LIN {X 0,Y 464.947,Z 367.068,A -85,B 0,C 180,E1 22700.512,E2 22700.512} C_VEL
LIN {X 0,Y 464.933,Z 367.036,A -85,B 0,C 180,E1 22696.87,E2 22696.87} C_VEL
LIN {X 0,Y 464.97,Z 367.067,A -85,B 0,C 180,E1 22693.422,E2 22693.422} C_VEL
LIN {X 0,Y 464.989,Z 367.031,A -85,B 0,C 180,E1 22689.774,E2 22689.774} C_VEL
LIN {X 0,Y 464.946,Z 367.064,A -85,B 0,C 180,E1 22686.291,E2 22686.291} C_VEL
LIN {X 0,Y 464.937,Z 367.047,A -85,B 0,C 180,E1 22682.706,E2 22682.706} C_VEL
LIN {X 0,Y 464.965,Z 367.06,A -85,B 0,C 180,E1 22679.132,E2 22679.132} C_VEL
LIN {X 0,Y 464.99,Z 367.048,A -85,B 0,C 180,E1 22675.555,E2 22675.555} C_VEL
LIN {X 0,Y 464.944,Z 367.049,A -85,B 0,C 180,E1 22672.084,E2 22672.084} C_VEL
LIN {X 0,Y 464.94,Z 367.063,A -85,B 0,C 180,E1 22668.459,E2 22668.459} C_VEL
LIN {X 0,Y 464.965,Z 367.041,A -85,B 0,C 180,E1 22664.906,E2 22664.906} C_VEL
LIN {X 0,Y 464.994,Z 367.06,A -85,B 0,C 180,E1 22661.309,E2 22661.309} C_VEL
LIN {X 0,Y 464.95,Z 367.044,A -85,B 0,C 180,E1 22657.756,E2 22657.756} C_VEL
LIN {X 0,Y 464.943,Z 367.064,A -85,B 0,C 180,E1 22654.249,E2 22654.249} C_VEL
LIN {X 0,Y 464.978,Z 367.05,A -85,B 0,C 180,E1 22650.779,E2 22650.779} C_VEL
LIN {X 0,Y 464.984,Z 367.05,A -85,B 0,C 180,E1 22647.219,E2 22647.219} C_VEL
LIN {X 0,Y 464.945,Z 367.068,A -85,B 0,C 180,E1 22643.741,E2 22643.741} C_VEL
LIN {X 0,Y 464.947,Z 367.069,A -85,B 0,C 180,E1 22640.142,E2 22640.142} C_VEL
LIN {X 0,Y 464.987,Z 367.066,A -85,B 0,C 180,E1 22636.617,E2 22636.617} C_VEL
LIN {X 0,Y 464.986,Z 367.052,A -85,B 0,C 180,E1 22632.971,E2 22632.971} C_VEL
LIN {X 0,Y 464.98,Z 367.258,A -85,B 0,C 180,E1 22631.366,E2 22631.366} C_VEL
LIN {X 0,Y 469.561,Z 382.374,A -85,B 0,C 180,E1 22628.405,E2 22628.405} C_VEL
LIN {X 0,Y 472.417,Z 392.249,A -85,B 0,C 180,E1 22626.661,E2 22626.661} C_VEL
LIN {X 0,Y 477.627,Z 402.671,A -85,B 0,C 180,E1 22626.002,E2 22626.002} C_VEL
LIN {X 0,Y 483.965,Z 427.071,A -85,B 0,C 180,E1 22625.03,E2 22625.03} C_VEL
LIN {X 0,Y 480.044,Z 648.164,A -85,B 0,C 180,E1 22621.453,E2 22621.453} C_VEL
LIN {X 0,Y 479.301,Z 666.693,A -85,B 0,C 180,E1 22621.018,E2 22621.018} C_VEL
LIN {X 0,Y 478.11,Z 687.493,A -85,B 0,C 180,E1 22620.307,E2 22620.307} C_VEL
LIN {X 0,Y 476.875,Z 704.905,A -85,B 0,C 180,E1 22619.519,E2 22619.519} C_VEL
LIN {X 0,Y 475.534,Z 721.763,A -85,B 0,C 180,E1 22618.581,E2 22618.581} C_VEL
LIN {X 0,Y 473.78,Z 741.15,A -85,B 0,C 180,E1 22617.254,E2 22617.254} C_VEL
LIN {X 0,Y 472.31,Z 756.498,A -85,B 0,C 180,E1 22615.989,E2 22615.989} C_VEL
LIN {X 0,Y 470.857,Z 771.086,A -85,B 0,C 180,E1 22614.594,E2 22614.594} C_VEL
LIN {X 0,Y 469.132,Z 788.25,A -85,B 0,C 180,E1 22612.65,E2 22612.65} C_VEL
LIN {X 0,Y 467.883,Z 800.978,A -85,B 0,C 180,E1 22610.951,E2 22610.951} C_VEL
LIN {X 0,Y 466.724,Z 813.64,A -85,B 0,C 180,E1 22609.003,E2 22609.003} C_VEL
LIN {X 0,Y 465.696,Z 825.892,A -85,B 0,C 180,E1 22606.745,E2 22606.745} C_VEL
LIN {X 0,Y 465.054,Z 834.762,A -85,B 0,C 180,E1 22604.823,E2 22604.823} C_VEL
LIN {X 0,Y 464.527,Z 843.637,A -85,B 0,C 180,E1 22602.556,E2 22602.556} C_VEL
LIN {X 0,Y 464.18,Z 851.15,A -85,B 0,C 180,E1 22600.129,E2 22600.129} C_VEL
LIN {X 0,Y 464.022,Z 856.246,A -85,B 0,C 180,E1 22598.051,E2 22598.051} C_VEL
LIN {X 0,Y 463.947,Z 860.214,A -85,B 0,C 180,E1 22595.937,E2 22595.937} C_VEL
LIN {X 0,Y 463.913,Z 863.438,A -85,B 0,C 180,E1 22593.336,E2 22593.336} C_VEL
LIN {X 0,Y 463.91,Z 864.696,A -85,B 0,C 180,E1 22591.111,E2 22591.111} C_VEL
LIN {X 0,Y 463.91,Z 864.755,A -85,B 0,C 180,E1 22589.136,E2 22589.136} C_VEL
LIN {X 0,Y 463.914,Z 863.704,A -85,B 0,C 180,E1 22587.035,E2 22587.035} C_VEL
LIN {X 0,Y 463.935,Z 861.041,A -85,B 0,C 180,E1 22584.559,E2 22584.559} C_VEL
LIN {X 0,Y 464.016,Z 856.788,A -85,B 0,C 180,E1 22582.198,E2 22582.198} C_VEL
LIN {X 0,Y 464.154,Z 852.036,A -85,B 0,C 180,E1 22580.202,E2 22580.202} C_VEL
LIN {X 0,Y 464.42,Z 845.709,A -85,B 0,C 180,E1 22578.072,E2 22578.072} C_VEL
LIN {X 0,Y 464.954,Z 836.391,A -85,B 0,C 180,E1 22575.555,E2 22575.555} C_VEL
LIN {X 0,Y 465.589,Z 827.257,A -85,B 0,C 180,E1 22573.533,E2 22573.533} C_VEL
LIN {X 0,Y 466.4,Z 817.262,A -85,B 0,C 180,E1 22571.632,E2 22571.632} C_VEL
LIN {X 0,Y 467.614,Z 803.952,A -85,B 0,C 180,E1 22569.473,E2 22569.473} C_VEL
LIN {X 0,Y 468.852,Z 790.947,A -85,B 0,C 180,E1 22567.692,E2 22567.692} C_VEL
LIN {X 0,Y 470.182,Z 777.792,A -85,B 0,C 180,E1 22566.126,E2 22566.126} C_VEL
LIN {X 0,Y 471.902,Z 760.777,A -85,B 0,C 180,E1 22564.392,E2 22564.392} C_VEL
LIN {X 0,Y 473.431,Z 744.821,A -85,B 0,C 180,E1 22563.033,E2 22563.033} C_VEL
LIN {X 0,Y 474.846,Z 729.536,A -85,B 0,C 180,E1 22561.92,E2 22561.92} C_VEL
LIN {X 0,Y 476.477,Z 710.731,A -85,B 0,C 180,E1 22560.777,E2 22560.777} C_VEL
LIN {X 0,Y 477.784,Z 692.136,A -85,B 0,C 180,E1 22559.887,E2 22559.887} C_VEL
LIN {X 0,Y 478.841,Z 675.18,A -85,B 0,C 180,E1 22559.246,E2 22559.246} C_VEL
LIN {X 0,Y 479.873,Z 654.59,A -85,B 0,C 180,E1 22558.671,E2 22558.671} C_VEL
LIN {X 0,Y 480.66,Z 617.37,A -85,B 0,C 180,E1 22558.034,E2 22558.034} C_VEL
LIN {X 0,Y 483.896,Z 426.069,A -85,B 0,C 180,E1 22554.947,E2 22554.947} C_VEL
LIN {X 0,Y 476.986,Z 401.05,A -85,B 0,C 180,E1 22553.913,E2 22553.913} C_VEL
LIN {X 0,Y 472.254,Z 391.785,A -85,B 0,C 180,E1 22553.289,E2 22553.289} C_VEL
LIN {X 0,Y 467.71,Z 376.233,A -85,B 0,C 180,E1 22550.429,E2 22550.429} C_VEL
LIN {X 0,Y 464.964,Z 367.167,A -85,B 0,C 180,E1 22548.586,E2 22548.586} C_VEL
LIN {X 0,Y 464.988,Z 367.054,A -85,B 0,C 180,E1 22545.031,E2 22545.031} C_VEL
LIN {X 0,Y 464.973,Z 367.053,A -85,B 0,C 180,E1 22541.48,E2 22541.48} C_VEL
LIN {X 0,Y 464.942,Z 367.054,A -85,B 0,C 180,E1 22537.959,E2 22537.959} C_VEL
LIN {X 0,Y 464.946,Z 367.058,A -85,B 0,C 180,E1 22534.297,E2 22534.297} C_VEL
LIN {X 0,Y 464.99,Z 367.066,A -85,B 0,C 180,E1 22530.785,E2 22530.785} C_VEL
LIN {X 0,Y 464.969,Z 367.038,A -85,B 0,C 180,E1 22527.264,E2 22527.264} C_VEL
LIN {X 0,Y 464.941,Z 367.065,A -85,B 0,C 180,E1 22523.716,E2 22523.716} C_VEL
LIN {X 0,Y 464.943,Z 367.055,A -85,B 0,C 180,E1 22519.992,E2 22519.992} C_VEL
LIN {X 0,Y 464.977,Z 367.056,A -85,B 0,C 180,E1 22516.459,E2 22516.459} C_VEL
LIN {X 0,Y 464.964,Z 367.04,A -85,B 0,C 180,E1 22513.054,E2 22513.054} C_VEL
LIN {X 0,Y 464.939,Z 367.066,A -85,B 0,C 180,E1 22509.536,E2 22509.536} C_VEL
LIN {X 0,Y 464.945,Z 367.037,A -85,B 0,C 180,E1 22505.93,E2 22505.93} C_VEL
LIN {X 0,Y 464.988,Z 367.066,A -85,B 0,C 180,E1 22502.347,E2 22502.347} C_VEL
LIN {X 0,Y 464.954,Z 367.035,A -85,B 0,C 180,E1 22498.896,E2 22498.896} C_VEL
LIN {X 0,Y 464.94,Z 367.065,A -85,B 0,C 180,E1 22495.318,E2 22495.318} C_VEL
LIN {X 0,Y 464.948,Z 367.043,A -85,B 0,C 180,E1 22491.722,E2 22491.722} C_VEL
LIN {X 0,Y 464.992,Z 367.054,A -85,B 0,C 180,E1 22488.219,E2 22488.219} C_VEL
LIN {X 0,Y 464.957,Z 367.054,A -85,B 0,C 180,E1 22484.669,E2 22484.669} C_VEL
LIN {X 0,Y 464.936,Z 367.06,A -85,B 0,C 180,E1 22481.121,E2 22481.121} C_VEL
LIN {X 0,Y 464.948,Z 367.053,A -85,B 0,C 180,E1 22477.501,E2 22477.501} C_VEL
LIN {X 0,Y 464.992,Z 367.055,A -85,B 0,C 180,E1 22473.99,E2 22473.99} C_VEL
LIN {X 0,Y 464.954,Z 367.067,A -85,B 0,C 180,E1 22470.507,E2 22470.507} C_VEL
LIN {X 0,Y 464.937,Z 367.068,A -85,B 0,C 180,E1 22466.9,E2 22466.9} C_VEL
LIN {X 0,Y 464.95,Z 367.067,A -85,B 0,C 180,E1 22463.295,E2 22463.295} C_VEL
LIN {X 0,Y 464.999,Z 367.064,A -85,B 0,C 180,E1 22459.757,E2 22459.757} C_VEL
LIN {X 0,Y 464.968,Z 367.069,A -85,B 0,C 180,E1 22456.084,E2 22456.084} C_VEL
LIN {X 0,Y 464.936,Z 367.069,A -85,B 0,C 180,E1 22452.64,E2 22452.64} C_VEL
LIN {X 0,Y 464.948,Z 367.067,A -85,B 0,C 180,E1 22449.055,E2 22449.055} C_VEL
LIN {X 0,Y 464.987,Z 367.065,A -85,B 0,C 180,E1 22445.49,E2 22445.49} C_VEL
LIN {X 0,Y 464.965,Z 367.067,A -85,B 0,C 180,E1 22441.87,E2 22441.87} C_VEL
LIN {X 0,Y 464.937,Z 367.068,A -85,B 0,C 180,E1 22438.376,E2 22438.376} C_VEL
LIN {X 0,Y 464.939,Z 367.07,A -85,B 0,C 180,E1 22434.657,E2 22434.657} C_VEL
LIN {X 0,Y 464.983,Z 367.067,A -85,B 0,C 180,E1 22431.176,E2 22431.176} C_VEL
LIN {X 0,Y 464.972,Z 367.067,A -85,B 0,C 180,E1 22429.595,E2 22429.595} C_VEL
LIN {X 0,Y 464.033,Z 367.192,A -85,B 0,C 180,E1 22428.646,E2 22428.646} C_VEL
LIN {X 0,Y 457.477,Z 368.001,A -85,B 0,C 180,E1 22425.906,E2 22425.906} C_VEL
LIN {X 0,Y 457.055,Z 368.052,A -85,B 0,C 180,E1 22425.278,E2 22425.278} C_VEL
LIN {X 0,Y 457.018,Z 368.057,A -85,B 0,C 180,E1 22421.611,E2 22421.611} C_VEL
LIN {X 0,Y 456.994,Z 368.06,A -85,B 0,C 180,E1 22418.049,E2 22418.049} C_VEL
LIN {X 0,Y 457.001,Z 368.057,A -85,B 0,C 180,E1 22414.392,E2 22414.392} C_VEL
LIN {X 0,Y 457.045,Z 368.053,A -85,B 0,C 180,E1 22410.877,E2 22410.877} C_VEL
LIN {X 0,Y 457.028,Z 368.055,A -85,B 0,C 180,E1 22407.241,E2 22407.241} C_VEL
LIN {X 0,Y 456.996,Z 368.059,A -85,B 0,C 180,E1 22403.72,E2 22403.72} C_VEL
LIN {X 0,Y 456.997,Z 368.059,A -85,B 0,C 180,E1 22400.047,E2 22400.047} C_VEL
LIN {X 0,Y 457.027,Z 368.055,A -85,B 0,C 180,E1 22396.463,E2 22396.463} C_VEL
LIN {X 0,Y 457.04,Z 368.054,A -85,B 0,C 180,E1 22392.911,E2 22392.911} C_VEL
LIN {X 0,Y 457.001,Z 368.056,A -85,B 0,C 180,E1 22389.376,E2 22389.376} C_VEL
LIN {X 0,Y 456.997,Z 368.059,A -85,B 0,C 180,E1 22385.713,E2 22385.713} C_VEL
LIN {X 0,Y 457.017,Z 368.057,A -85,B 0,C 180,E1 22382.084,E2 22382.084} C_VEL
LIN {X 0,Y 457.055,Z 368.054,A -85,B 0,C 180,E1 22378.541,E2 22378.541} C_VEL
LIN {X 0,Y 457.019,Z 368.057,A -85,B 0,C 180,E1 22374.874,E2 22374.874} C_VEL
LIN {X 0,Y 456.997,Z 368.057,A -85,B 0,C 180,E1 22371.265,E2 22371.265} C_VEL
LIN {X 0,Y 457.006,Z 368.058,A -85,B 0,C 180,E1 22367.636,E2 22367.636} C_VEL
LIN {X 0,Y 457.042,Z 368.055,A -85,B 0,C 180,E1 22364.07,E2 22364.07} C_VEL
LIN {X 0,Y 457.048,Z 368.054,A -85,B 0,C 180,E1 22360.346,E2 22360.346} C_VEL
LIN {X 0,Y 457.005,Z 368.056,A -85,B 0,C 180,E1 22356.8,E2 22356.8} C_VEL
LIN {X 0,Y 456.999,Z 368.058,A -85,B 0,C 180,E1 22353.15,E2 22353.15} C_VEL
LIN {X 0,Y 457.025,Z 368.056,A -85,B 0,C 180,E1 22349.624,E2 22349.624} C_VEL
LIN {X 0,Y 457.049,Z 368.045,A -85,B 0,C 180,E1 22346.078,E2 22346.078} C_VEL
LIN {X 0,Y 457.01,Z 368.042,A -85,B 0,C 180,E1 22342.504,E2 22342.504} C_VEL
LIN {X 0,Y 456.998,Z 368.048,A -85,B 0,C 180,E1 22338.886,E2 22338.886} C_VEL
LIN {X 0,Y 457.011,Z 368.044,A -85,B 0,C 180,E1 22335.247,E2 22335.247} C_VEL
LIN {X 0,Y 457.053,Z 368.041,A -85,B 0,C 180,E1 22331.732,E2 22331.732} C_VEL
LIN {X 0,Y 457.025,Z 368.031,A -85,B 0,C 180,E1 22328.043,E2 22328.043} C_VEL
LIN {X 0,Y 457.001,Z 368.054,A -85,B 0,C 180,E1 22324.512,E2 22324.512} C_VEL
LIN {X 0,Y 456.999,Z 368.028,A -85,B 0,C 180,E1 22320.747,E2 22320.747} C_VEL
LIN {X 0,Y 457.039,Z 368.053,A -85,B 0,C 180,E1 22317.236,E2 22317.236} C_VEL
LIN {X 0,Y 457.046,Z 368.017,A -85,B 0,C 180,E1 22313.589,E2 22313.589} C_VEL
LIN {X 0,Y 457.009,Z 368.055,A -85,B 0,C 180,E1 22310.042,E2 22310.042} C_VEL
LIN {X 0,Y 457,Z 368.027,A -85,B 0,C 180,E1 22306.457,E2 22306.457} C_VEL
LIN {X 0,Y 457.034,Z 368.056,A -85,B 0,C 180,E1 22302.941,E2 22302.941} C_VEL
LIN {X 0,Y 457.058,Z 368.022,A -85,B 0,C 180,E1 22299.24,E2 22299.24} C_VEL
LIN {X 0,Y 457.015,Z 368.055,A -85,B 0,C 180,E1 22295.709,E2 22295.709} C_VEL
LIN {X 0,Y 457,Z 368.026,A -85,B 0,C 180,E1 22292.078,E2 22292.078} C_VEL
LIN {X 0,Y 457.017,Z 368.053,A -85,B 0,C 180,E1 22288.47,E2 22288.47} C_VEL
LIN {X 0,Y 457.052,Z 368.052,A -85,B 0,C 180,E1 22284.872,E2 22284.872} C_VEL
LIN {X 0,Y 457.032,Z 368.045,A -85,B 0,C 180,E1 22281.264,E2 22281.264} C_VEL
LIN {X 0,Y 457.006,Z 368.05,A -85,B 0,C 180,E1 22277.686,E2 22277.686} C_VEL
LIN {X 0,Y 457.006,Z 368.061,A -85,B 0,C 180,E1 22273.91,E2 22273.91} C_VEL
LIN {X 0,Y 457.037,Z 368.25,A -85,B 0,C 180,E1 22272.022,E2 22272.022} C_VEL
LIN {X 0,Y 461.532,Z 382.762,A -85,B 0,C 180,E1 22269.08,E2 22269.08} C_VEL
LIN {X 0,Y 464.235,Z 391.951,A -85,B 0,C 180,E1 22267.416,E2 22267.416} C_VEL
LIN {X 0,Y 471.676,Z 406.668,A -85,B 0,C 180,E1 22266.451,E2 22266.451} C_VEL
LIN {X 0,Y 477.373,Z 428.874,A -85,B 0,C 180,E1 22265.549,E2 22265.549} C_VEL
LIN {X 0,Y 473.204,Z 648.338,A -85,B 0,C 180,E1 22261.952,E2 22261.952} C_VEL
LIN {X 0,Y 472.379,Z 667.608,A -85,B 0,C 180,E1 22261.49,E2 22261.49} C_VEL
LIN {X 0,Y 471.092,Z 688.176,A -85,B 0,C 180,E1 22260.763,E2 22260.763} C_VEL
LIN {X 0,Y 469.847,Z 704.666,A -85,B 0,C 180,E1 22260.005,E2 22260.005} C_VEL
LIN {X 0,Y 468.407,Z 721.599,A -85,B 0,C 180,E1 22259.052,E2 22259.052} C_VEL
LIN {X 0,Y 466.547,Z 740.909,A -85,B 0,C 180,E1 22257.713,E2 22257.713} C_VEL
LIN {X 0,Y 464.968,Z 756.256,A -85,B 0,C 180,E1 22256.431,E2 22256.431} C_VEL
LIN {X 0,Y 463.362,Z 771.413,A -85,B 0,C 180,E1 22254.958,E2 22254.958} C_VEL
LIN {X 0,Y 461.598,Z 787.697,A -85,B 0,C 180,E1 22253.082,E2 22253.082} C_VEL
LIN {X 0,Y 460.272,Z 800.136,A -85,B 0,C 180,E1 22251.404,E2 22251.404} C_VEL
LIN {X 0,Y 459.109,Z 811.808,A -85,B 0,C 180,E1 22249.595,E2 22249.595} C_VEL
LIN {X 0,Y 457.949,Z 824.531,A -85,B 0,C 180,E1 22247.273,E2 22247.273} C_VEL
LIN {X 0,Y 457.19,Z 833.977,A -85,B 0,C 180,E1 22245.214,E2 22245.214} C_VEL
LIN {X 0,Y 456.655,Z 841.986,A -85,B 0,C 180,E1 22243.162,E2 22243.162} C_VEL
LIN {X 0,Y 456.223,Z 850.457,A -85,B 0,C 180,E1 22240.48,E2 22240.48} C_VEL
LIN {X 0,Y 456.042,Z 855.737,A -85,B 0,C 180,E1 22238.32,E2 22238.32} C_VEL
LIN {X 0,Y 455.952,Z 859.559,A -85,B 0,C 180,E1 22236.295,E2 22236.295} C_VEL
LIN {X 0,Y 455.918,Z 862.746,A -85,B 0,C 180,E1 22233.898,E2 22233.898} C_VEL
LIN {X 0,Y 455.91,Z 864.43,A -85,B 0,C 180,E1 22231.257,E2 22231.257} C_VEL
LIN {X 0,Y 455.914,Z 864.519,A -85,B 0,C 180,E1 22229.12,E2 22229.12} C_VEL
LIN {X 0,Y 455.916,Z 863.468,A -85,B 0,C 180,E1 22226.983,E2 22226.983} C_VEL
LIN {X 0,Y 455.938,Z 860.804,A -85,B 0,C 180,E1 22224.463,E2 22224.463} C_VEL
LIN {X 0,Y 456.018,Z 856.549,A -85,B 0,C 180,E1 22222.06,E2 22222.06} C_VEL
LIN {X 0,Y 456.168,Z 851.796,A -85,B 0,C 180,E1 22220.029,E2 22220.029} C_VEL
LIN {X 0,Y 456.438,Z 845.869,A -85,B 0,C 180,E1 22217.989,E2 22217.989} C_VEL
LIN {X 0,Y 456.976,Z 837.236,A -85,B 0,C 180,E1 22215.557,E2 22215.557} C_VEL
LIN {X 0,Y 457.682,Z 827.636,A -85,B 0,C 180,E1 22213.371,E2 22213.371} C_VEL
LIN {X 0,Y 458.545,Z 817.723,A -85,B 0,C 180,E1 22211.437,E2 22211.437} C_VEL
LIN {X 0,Y 459.756,Z 805.452,A -85,B 0,C 180,E1 22209.372,E2 22209.372} C_VEL
LIN {X 0,Y 461.208,Z 791.206,A -85,B 0,C 180,E1 22207.369,E2 22207.369} C_VEL
LIN {X 0,Y 462.606,Z 778.299,A -85,B 0,C 180,E1 22205.8,E2 22205.8} C_VEL
LIN {X 0,Y 464.398,Z 761.956,A -85,B 0,C 180,E1 22204.084,E2 22204.084} C_VEL
LIN {X 0,Y 466.124,Z 745.03,A -85,B 0,C 180,E1 22202.613,E2 22202.613} C_VEL
LIN {X 0,Y 467.611,Z 730.042,A -85,B 0,C 180,E1 22201.503,E2 22201.503} C_VEL
LIN {X 0,Y 469.293,Z 712.008,A -85,B 0,C 180,E1 22200.377,E2 22200.377} C_VEL
LIN {X 0,Y 470.764,Z 692.642,A -85,B 0,C 180,E1 22199.425,E2 22199.425} C_VEL
LIN {X 0,Y 471.897,Z 675.635,A -85,B 0,C 180,E1 22198.77,E2 22198.77} C_VEL
LIN {X 0,Y 472.955,Z 656.127,A -85,B 0,C 180,E1 22198.207,E2 22198.207} C_VEL
LIN {X 0,Y 473.71,Z 626.054,A -85,B 0,C 180,E1 22197.664,E2 22197.664} C_VEL
LIN {X 0,Y 477.298,Z 427.781,A -85,B 0,C 180,E1 22194.425,E2 22194.425} C_VEL
LIN {X 0,Y 471.128,Z 405.209,A -85,B 0,C 180,E1 22193.473,E2 22193.473} C_VEL
LIN {X 0,Y 464.067,Z 391.471,A -85,B 0,C 180,E1 22192.535,E2 22192.535} C_VEL
LIN {X 0,Y 459.441,Z 375.913,A -85,B 0,C 180,E1 22189.571,E2 22189.571} C_VEL
LIN {X 0,Y 457.024,Z 368.144,A -85,B 0,C 180,E1 22187.934,E2 22187.934} C_VEL
LIN {X 0,Y 457.005,Z 368.05,A -85,B 0,C 180,E1 22184.264,E2 22184.264} C_VEL
LIN {X 0,Y 457.026,Z 368.049,A -85,B 0,C 180,E1 22180.692,E2 22180.692} C_VEL
LIN {X 0,Y 457.055,Z 368.038,A -85,B 0,C 180,E1 22177.145,E2 22177.145} C_VEL
LIN {X 0,Y 457.022,Z 368.038,A -85,B 0,C 180,E1 22173.461,E2 22173.461} C_VEL
LIN {X 0,Y 457.004,Z 368.054,A -85,B 0,C 180,E1 22169.927,E2 22169.927} C_VEL
LIN {X 0,Y 457.012,Z 368.048,A -85,B 0,C 180,E1 22166.232,E2 22166.232} C_VEL
LIN {X 0,Y 457.047,Z 368.032,A -85,B 0,C 180,E1 22162.65,E2 22162.65} C_VEL
LIN {X 0,Y 457.04,Z 368.046,A -85,B 0,C 180,E1 22159.028,E2 22159.028} C_VEL
LIN {X 0,Y 457.003,Z 368.039,A -85,B 0,C 180,E1 22155.486,E2 22155.486} C_VEL
LIN {X 0,Y 457.001,Z 368.052,A -85,B 0,C 180,E1 22151.745,E2 22151.745} C_VEL
LIN {X 0,Y 457.023,Z 368.037,A -85,B 0,C 180,E1 22148.18,E2 22148.18} C_VEL
LIN {X 0,Y 457.048,Z 368.033,A -85,B 0,C 180,E1 22144.648,E2 22144.648} C_VEL
LIN {X 0,Y 457.016,Z 368.053,A -85,B 0,C 180,E1 22141.008,E2 22141.008} C_VEL
LIN {X 0,Y 456.997,Z 368.032,A -85,B 0,C 180,E1 22137.372,E2 22137.372} C_VEL
LIN {X 0,Y 457.008,Z 368.053,A -85,B 0,C 180,E1 22133.726,E2 22133.726} C_VEL
LIN {X 0,Y 457.046,Z 368.018,A -85,B 0,C 180,E1 22130.181,E2 22130.181} C_VEL
LIN {X 0,Y 457.042,Z 368.056,A -85,B 0,C 180,E1 22126.469,E2 22126.469} C_VEL
LIN {X 0,Y 456.999,Z 368.022,A -85,B 0,C 180,E1 22122.955,E2 22122.955} C_VEL
LIN {X 0,Y 457,Z 368.057,A -85,B 0,C 180,E1 22119.249,E2 22119.249} C_VEL
LIN {X 0,Y 457.026,Z 368.027,A -85,B 0,C 180,E1 22115.722,E2 22115.722} C_VEL
LIN {X 0,Y 457.057,Z 368.055,A -85,B 0,C 180,E1 22112.094,E2 22112.094} C_VEL
LIN {X 0,Y 457.009,Z 368.057,A -85,B 0,C 180,E1 22108.565,E2 22108.565} C_VEL
LIN {X 0,Y 456.999,Z 368.058,A -85,B 0,C 180,E1 22104.909,E2 22104.909} C_VEL
LIN {X 0,Y 457.01,Z 368.056,A -85,B 0,C 180,E1 22101.275,E2 22101.275} C_VEL
LIN {X 0,Y 457.052,Z 368.054,A -85,B 0,C 180,E1 22097.82,E2 22097.82} C_VEL
LIN {X 0,Y 457.02,Z 368.057,A -85,B 0,C 180,E1 22094.156,E2 22094.156} C_VEL
LIN {X 0,Y 456.996,Z 368.057,A -85,B 0,C 180,E1 22090.62,E2 22090.62} C_VEL
LIN {X 0,Y 457.007,Z 368.057,A -85,B 0,C 180,E1 22086.987,E2 22086.987} C_VEL
LIN {X 0,Y 457.053,Z 368.053,A -85,B 0,C 180,E1 22083.454,E2 22083.454} C_VEL
LIN {X 0,Y 457.018,Z 368.056,A -85,B 0,C 180,E1 22079.921,E2 22079.921} C_VEL
LIN {X 0,Y 456.997,Z 368.059,A -85,B 0,C 180,E1 22076.368,E2 22076.368} C_VEL
LIN {X 0,Y 457,Z 368.059,A -85,B 0,C 180,E1 22072.647,E2 22072.647} C_VEL
LIN {X 0,Y 457.038,Z 368.055,A -85,B 0,C 180,E1 22069.105,E2 22069.105} C_VEL
LIN {X 0,Y 457.036,Z 368.055,A -85,B 0,C 180,E1 22065.479,E2 22065.479} C_VEL
LIN {X 0,Y 457.055,Z 368.052,A -85,B 0,C 180,E1 22065.278,E2 22065.278} C_VEL
LIN {X 0,Y 456.105,Z 368.174,A -85,B 0,C 180,E1 22064.313,E2 22064.313} C_VEL
LIN {X 0,Y 449.57,Z 368.988,A -85,B 0,C 180,E1 22061.527,E2 22061.527} C_VEL
LIN {X 0,Y 449.09,Z 369.044,A -85,B 0,C 180,E1 22060.888,E2 22060.888} C_VEL
LIN {X 0,Y 449.117,Z 369.041,A -85,B 0,C 180,E1 22057.162,E2 22057.162} C_VEL
LIN {X 0,Y 449.08,Z 369.046,A -85,B 0,C 180,E1 22053.446,E2 22053.446} C_VEL
LIN {X 0,Y 449.055,Z 369.05,A -85,B 0,C 180,E1 22049.872,E2 22049.872} C_VEL
LIN {X 0,Y 449.059,Z 369.046,A -85,B 0,C 180,E1 22046.17,E2 22046.17} C_VEL
LIN {X 0,Y 449.089,Z 369.044,A -85,B 0,C 180,E1 22042.581,E2 22042.581} C_VEL
LIN {X 0,Y 449.102,Z 369.044,A -85,B 0,C 180,E1 22038.962,E2 22038.962} C_VEL
LIN {X 0,Y 449.064,Z 369.048,A -85,B 0,C 180,E1 22035.428,E2 22035.428} C_VEL
LIN {X 0,Y 449.057,Z 369.048,A -85,B 0,C 180,E1 22031.703,E2 22031.703} C_VEL
LIN {X 0,Y 449.068,Z 369.046,A -85,B 0,C 180,E1 22028.035,E2 22028.035} C_VEL
LIN {X 0,Y 449.103,Z 369.044,A -85,B 0,C 180,E1 22024.412,E2 22024.412} C_VEL
LIN {X 0,Y 449.108,Z 369.044,A -85,B 0,C 180,E1 22020.674,E2 22020.674} C_VEL
LIN {X 0,Y 449.07,Z 369.048,A -85,B 0,C 180,E1 22017.06,E2 22017.06} C_VEL
LIN {X 0,Y 449.058,Z 369.047,A -85,B 0,C 180,E1 22013.366,E2 22013.366} C_VEL
LIN {X 0,Y 449.065,Z 369.045,A -85,B 0,C 180,E1 22009.616,E2 22009.616} C_VEL
LIN {X 0,Y 449.094,Z 369.044,A -85,B 0,C 180,E1 22006.004,E2 22006.004} C_VEL
LIN {X 0,Y 449.11,Z 369.042,A -85,B 0,C 180,E1 22002.344,E2 22002.344} C_VEL
LIN {X 0,Y 449.066,Z 369.045,A -85,B 0,C 180,E1 21998.807,E2 21998.807} C_VEL
LIN {X 0,Y 449.061,Z 369.047,A -85,B 0,C 180,E1 21995.202,E2 21995.202} C_VEL
LIN {X 0,Y 449.077,Z 369.046,A -85,B 0,C 180,E1 21991.54,E2 21991.54} C_VEL
LIN {X 0,Y 449.118,Z 369.044,A -85,B 0,C 180,E1 21988.009,E2 21988.009} C_VEL
LIN {X 0,Y 449.083,Z 369.015,A -85,B 0,C 180,E1 21984.316,E2 21984.316} C_VEL
LIN {X 0,Y 449.062,Z 369.046,A -85,B 0,C 180,E1 21980.752,E2 21980.752} C_VEL
LIN {X 0,Y 449.058,Z 369.01,A -85,B 0,C 180,E1 21976.952,E2 21976.952} C_VEL
LIN {X 0,Y 449.087,Z 369.045,A -85,B 0,C 180,E1 21973.365,E2 21973.365} C_VEL
LIN {X 0,Y 449.11,Z 369.005,A -85,B 0,C 180,E1 21969.735,E2 21969.735} C_VEL
LIN {X 0,Y 449.079,Z 369.042,A -85,B 0,C 180,E1 21966.129,E2 21966.129} C_VEL
LIN {X 0,Y 449.058,Z 369.018,A -85,B 0,C 180,E1 21962.547,E2 21962.547} C_VEL
LIN {X 0,Y 449.07,Z 369.042,A -85,B 0,C 180,E1 21958.846,E2 21958.846} C_VEL
LIN {X 0,Y 449.102,Z 369.021,A -85,B 0,C 180,E1 21955.27,E2 21955.27} C_VEL
LIN {X 0,Y 449.11,Z 369.025,A -85,B 0,C 180,E1 21951.546,E2 21951.546} C_VEL
LIN {X 0,Y 449.074,Z 369.035,A -85,B 0,C 180,E1 21947.914,E2 21947.914} C_VEL
LIN {X 0,Y 449.062,Z 369.029,A -85,B 0,C 180,E1 21944.366,E2 21944.366} C_VEL
LIN {X 0,Y 449.081,Z 369.034,A -85,B 0,C 180,E1 21940.732,E2 21940.732} C_VEL
LIN {X 0,Y 449.116,Z 369.023,A -85,B 0,C 180,E1 21937.066,E2 21937.066} C_VEL
LIN {X 0,Y 449.095,Z 369.024,A -85,B 0,C 180,E1 21933.412,E2 21933.412} C_VEL
LIN {X 0,Y 449.065,Z 369.043,A -85,B 0,C 180,E1 21929.932,E2 21929.932} C_VEL
LIN {X 0,Y 449.065,Z 369.03,A -85,B 0,C 180,E1 21926.147,E2 21926.147} C_VEL
LIN {X 0,Y 449.091,Z 369.027,A -85,B 0,C 180,E1 21922.565,E2 21922.565} C_VEL
LIN {X 0,Y 449.12,Z 369.029,A -85,B 0,C 180,E1 21918.944,E2 21918.944} C_VEL
LIN {X 0,Y 449.086,Z 369.033,A -85,B 0,C 180,E1 21915.252,E2 21915.252} C_VEL
LIN {X 0,Y 449.156,Z 369.304,A -85,B 0,C 180,E1 21912.679,E2 21912.679} C_VEL
LIN {X 0,Y 453.835,Z 384.39,A -85,B 0,C 180,E1 21909.544,E2 21909.544} C_VEL
LIN {X 0,Y 455.946,Z 391.591,A -85,B 0,C 180,E1 21908.219,E2 21908.219} C_VEL
LIN {X 0,Y 465.679,Z 410.336,A -85,B 0,C 180,E1 21906.925,E2 21906.925} C_VEL
LIN {X 0,Y 470.821,Z 430.6,A -85,B 0,C 180,E1 21906.085,E2 21906.085} C_VEL
LIN {X 0,Y 466.403,Z 648.409,A -85,B 0,C 180,E1 21902.468,E2 21902.468} C_VEL
LIN {X 0,Y 465.494,Z 668.433,A -85,B 0,C 180,E1 21901.978,E2 21901.978} C_VEL
LIN {X 0,Y 464.119,Z 688.682,A -85,B 0,C 180,E1 21901.241,E2 21901.241} C_VEL
LIN {X 0,Y 462.858,Z 704.427,A -85,B 0,C 180,E1 21900.506,E2 21900.506} C_VEL
LIN {X 0,Y 461.322,Z 721.359,A -85,B 0,C 180,E1 21899.542,E2 21899.542} C_VEL
LIN {X 0,Y 459.306,Z 741.044,A -85,B 0,C 180,E1 21898.155,E2 21898.155} C_VEL
LIN {X 0,Y 457.656,Z 756.015,A -85,B 0,C 180,E1 21896.887,E2 21896.887} C_VEL
LIN {X 0,Y 456.009,Z 770.602,A -85,B 0,C 180,E1 21895.451,E2 21895.451} C_VEL
LIN {X 0,Y 454.049,Z 787.454,A -85,B 0,C 180,E1 21893.489,E2 21893.489} C_VEL
LIN {X 0,Y 452.628,Z 799.893,A -85,B 0,C 180,E1 21891.784,E2 21891.784} C_VEL
LIN {X 0,Y 451.377,Z 811.565,A -85,B 0,C 180,E1 21889.945,E2 21889.945} C_VEL
LIN {X 0,Y 450.12,Z 824.288,A -85,B 0,C 180,E1 21887.583,E2 21887.583} C_VEL
LIN {X 0,Y 449.298,Z 833.735,A -85,B 0,C 180,E1 21885.488,E2 21885.488} C_VEL
LIN {X 0,Y 448.714,Z 841.745,A -85,B 0,C 180,E1 21883.399,E2 21883.399} C_VEL
LIN {X 0,Y 448.251,Z 850.217,A -85,B 0,C 180,E1 21880.669,E2 21880.669} C_VEL
LIN {X 0,Y 448.053,Z 855.498,A -85,B 0,C 180,E1 21878.469,E2 21878.469} C_VEL
LIN {X 0,Y 447.954,Z 859.321,A -85,B 0,C 180,E1 21876.408,E2 21876.408} C_VEL
LIN {X 0,Y 447.92,Z 862.51,A -85,B 0,C 180,E1 21873.968,E2 21873.968} C_VEL
LIN {X 0,Y 447.912,Z 864.194,A -85,B 0,C 180,E1 21871.279,E2 21871.279} C_VEL
LIN {X 0,Y 447.917,Z 864.283,A -85,B 0,C 180,E1 21869.105,E2 21869.105} C_VEL
LIN {X 0,Y 447.919,Z 863.231,A -85,B 0,C 180,E1 21866.929,E2 21866.929} C_VEL
LIN {X 0,Y 447.941,Z 860.566,A -85,B 0,C 180,E1 21864.364,E2 21864.364} C_VEL
LIN {X 0,Y 448.023,Z 856.31,A -85,B 0,C 180,E1 21861.918,E2 21861.918} C_VEL
LIN {X 0,Y 448.186,Z 851.557,A -85,B 0,C 180,E1 21859.849,E2 21859.849} C_VEL
LIN {X 0,Y 448.479,Z 845.629,A -85,B 0,C 180,E1 21857.773,E2 21857.773} C_VEL
LIN {X 0,Y 449.062,Z 836.995,A -85,B 0,C 180,E1 21855.296,E2 21855.296} C_VEL
LIN {X 0,Y 449.832,Z 827.393,A -85,B 0,C 180,E1 21853.072,E2 21853.072} C_VEL
LIN {X 0,Y 450.766,Z 817.481,A -85,B 0,C 180,E1 21851.105,E2 21851.105} C_VEL
LIN {X 0,Y 452.11,Z 804.895,A -85,B 0,C 180,E1 21848.955,E2 21848.955} C_VEL
LIN {X 0,Y 453.639,Z 790.963,A -85,B 0,C 180,E1 21846.97,E2 21846.97} C_VEL
LIN {X 0,Y 455.11,Z 778.241,A -85,B 0,C 180,E1 21845.398,E2 21845.398} C_VEL
LIN {X 0,Y 456.976,Z 762.38,A -85,B 0,C 180,E1 21843.701,E2 21843.701} C_VEL
LIN {X 0,Y 458.816,Z 745.517,A -85,B 0,C 180,E1 21842.203,E2 21842.203} C_VEL
LIN {X 0,Y 460.451,Z 730.066,A -85,B 0,C 180,E1 21841.038,E2 21841.038} C_VEL
LIN {X 0,Y 462.263,Z 711.779,A -85,B 0,C 180,E1 21839.881,E2 21839.881} C_VEL
LIN {X 0,Y 463.83,Z 692.403,A -85,B 0,C 180,E1 21838.918,E2 21838.918} C_VEL
LIN {X 0,Y 465.029,Z 675.472,A -85,B 0,C 180,E1 21838.259,E2 21838.259} C_VEL
LIN {X 0,Y 466.117,Z 656.39,A -85,B 0,C 180,E1 21837.7,E2 21837.7} C_VEL
LIN {X 0,Y 466.913,Z 627.601,A -85,B 0,C 180,E1 21837.167,E2 21837.167} C_VEL
LIN {X 0,Y 470.764,Z 429.657,A -85,B 0,C 180,E1 21833.893,E2 21833.893} C_VEL
LIN {X 0,Y 465.167,Z 409.085,A -85,B 0,C 180,E1 21833.005,E2 21833.005} C_VEL
LIN {X 0,Y 455.776,Z 391.131,A -85,B 0,C 180,E1 21831.732,E2 21831.732} C_VEL
LIN {X 0,Y 451.418,Z 376.528,A -85,B 0,C 180,E1 21828.861,E2 21828.861} C_VEL
LIN {X 0,Y 449.126,Z 369.099,A -85,B 0,C 180,E1 21827.236,E2 21827.236} C_VEL
LIN {X 0,Y 449.101,Z 369.044,A -85,B 0,C 180,E1 21823.467,E2 21823.467} C_VEL
LIN {X 0,Y 449.069,Z 369.047,A -85,B 0,C 180,E1 21819.888,E2 21819.888} C_VEL
LIN {X 0,Y 449.066,Z 369.047,A -85,B 0,C 180,E1 21816.163,E2 21816.163} C_VEL
LIN {X 0,Y 449.09,Z 369.03,A -85,B 0,C 180,E1 21812.605,E2 21812.605} C_VEL
LIN {X 0,Y 449.124,Z 369.016,A -85,B 0,C 180,E1 21808.968,E2 21808.968} C_VEL
LIN {X 0,Y 449.086,Z 369.041,A -85,B 0,C 180,E1 21805.312,E2 21805.312} C_VEL
LIN {X 0,Y 449.062,Z 369.015,A -85,B 0,C 180,E1 21801.696,E2 21801.696} C_VEL
LIN {X 0,Y 449.064,Z 369.045,A -85,B 0,C 180,E1 21797.899,E2 21797.899} C_VEL
LIN {X 0,Y 449.086,Z 369.008,A -85,B 0,C 180,E1 21794.313,E2 21794.313} C_VEL
LIN {X 0,Y 449.114,Z 369.042,A -85,B 0,C 180,E1 21790.653,E2 21790.653} C_VEL
LIN {X 0,Y 449.077,Z 369.011,A -85,B 0,C 180,E1 21787.039,E2 21787.039} C_VEL
LIN {X 0,Y 449.061,Z 369.042,A -85,B 0,C 180,E1 21783.452,E2 21783.452} C_VEL
LIN {X 0,Y 449.063,Z 369.022,A -85,B 0,C 180,E1 21779.75,E2 21779.75} C_VEL
LIN {X 0,Y 449.1,Z 369.03,A -85,B 0,C 180,E1 21776.176,E2 21776.176} C_VEL
LIN {X 0,Y 449.112,Z 369.023,A -85,B 0,C 180,E1 21772.458,E2 21772.458} C_VEL
LIN {X 0,Y 449.073,Z 369.028,A -85,B 0,C 180,E1 21768.837,E2 21768.837} C_VEL
LIN {X 0,Y 449.059,Z 369.04,A -85,B 0,C 180,E1 21765.303,E2 21765.303} C_VEL
LIN {X 0,Y 449.079,Z 369.021,A -85,B 0,C 180,E1 21761.711,E2 21761.711} C_VEL
LIN {X 0,Y 449.122,Z 369.03,A -85,B 0,C 180,E1 21758.044,E2 21758.044} C_VEL
LIN {X 0,Y 449.098,Z 369.029,A -85,B 0,C 180,E1 21754.277,E2 21754.277} C_VEL
LIN {X 0,Y 449.068,Z 369.046,A -85,B 0,C 180,E1 21750.679,E2 21750.679} C_VEL
LIN {X 0,Y 449.06,Z 369.047,A -85,B 0,C 180,E1 21746.95,E2 21746.95} C_VEL
LIN {X 0,Y 449.071,Z 369.045,A -85,B 0,C 180,E1 21743.275,E2 21743.275} C_VEL
LIN {X 0,Y 449.122,Z 369.042,A -85,B 0,C 180,E1 21739.781,E2 21739.781} C_VEL
LIN {X 0,Y 449.099,Z 369.044,A -85,B 0,C 180,E1 21735.98,E2 21735.98} C_VEL
LIN {X 0,Y 449.066,Z 369.047,A -85,B 0,C 180,E1 21732.349,E2 21732.349} C_VEL
LIN {X 0,Y 449.059,Z 369.045,A -85,B 0,C 180,E1 21728.73,E2 21728.73} C_VEL
LIN {X 0,Y 449.087,Z 369.045,A -85,B 0,C 180,E1 21725.214,E2 21725.214} C_VEL
LIN {X 0,Y 449.118,Z 369.042,A -85,B 0,C 180,E1 21721.515,E2 21721.515} C_VEL
LIN {X 0,Y 449.081,Z 369.046,A -85,B 0,C 180,E1 21717.875,E2 21717.875} C_VEL
LIN {X 0,Y 449.059,Z 369.049,A -85,B 0,C 180,E1 21714.324,E2 21714.324} C_VEL
LIN {X 0,Y 449.061,Z 369.046,A -85,B 0,C 180,E1 21710.597,E2 21710.597} C_VEL
LIN {X 0,Y 449.088,Z 369.044,A -85,B 0,C 180,E1 21706.957,E2 21706.957} C_VEL
LIN {X 0,Y 449.103,Z 369.043,A -85,B 0,C 180,E1 21703.387,E2 21703.387} C_VEL
LIN {X 0,Y 449.09,Z 369.044,A -85,B 0,C 180,E1 21700.888,E2 21700.888} C_VEL
LIN {X 0,Y 448.058,Z 369.174,A -85,B 0,C 180,E1 21699.906,E2 21699.906} C_VEL
LIN {X 0,Y 441.576,Z 369.984,A -85,B 0,C 180,E1 21697.068,E2 21697.068} C_VEL
LIN {X 0,Y 441.124,Z 370.038,A -85,B 0,C 180,E1 21696.418,E2 21696.418} C_VEL
LIN {X 0,Y 441.158,Z 370.033,A -85,B 0,C 180,E1 21692.858,E2 21692.858} C_VEL
LIN {X 0,Y 441.169,Z 370.031,A -85,B 0,C 180,E1 21689.091,E2 21689.091} C_VEL
LIN {X 0,Y 441.141,Z 370.035,A -85,B 0,C 180,E1 21685.32,E2 21685.32} C_VEL
LIN {X 0,Y 441.117,Z 370.039,A -85,B 0,C 180,E1 21681.79,E2 21681.79} C_VEL
LIN {X 0,Y 441.12,Z 370.035,A -85,B 0,C 180,E1 21677.964,E2 21677.964} C_VEL
LIN {X 0,Y 441.142,Z 370.034,A -85,B 0,C 180,E1 21674.353,E2 21674.353} C_VEL
LIN {X 0,Y 441.173,Z 370.033,A -85,B 0,C 180,E1 21670.678,E2 21670.678} C_VEL
LIN {X 0,Y 441.152,Z 370.036,A -85,B 0,C 180,E1 21666.929,E2 21666.929} C_VEL
LIN {X 0,Y 441.128,Z 370.036,A -85,B 0,C 180,E1 21663.237,E2 21663.237} C_VEL
LIN {X 0,Y 441.119,Z 370.035,A -85,B 0,C 180,E1 21659.639,E2 21659.639} C_VEL
LIN {X 0,Y 441.144,Z 370.035,A -85,B 0,C 180,E1 21656.036,E2 21656.036} C_VEL
LIN {X 0,Y 441.17,Z 370.034,A -85,B 0,C 180,E1 21652.261,E2 21652.261} C_VEL
LIN {X 0,Y 441.16,Z 370.035,A -85,B 0,C 180,E1 21648.564,E2 21648.564} C_VEL
LIN {X 0,Y 441.127,Z 370.037,A -85,B 0,C 180,E1 21644.994,E2 21644.994} C_VEL
LIN {X 0,Y 441.119,Z 370.036,A -85,B 0,C 180,E1 21641.258,E2 21641.258} C_VEL
LIN {X 0,Y 441.143,Z 370.033,A -85,B 0,C 180,E1 21637.721,E2 21637.721} C_VEL
LIN {X 0,Y 441.171,Z 370.034,A -85,B 0,C 180,E1 21634.032,E2 21634.032} C_VEL
LIN {X 0,Y 441.158,Z 370.035,A -85,B 0,C 180,E1 21630.29,E2 21630.29} C_VEL
LIN {X 0,Y 441.128,Z 370.036,A -85,B 0,C 180,E1 21626.657,E2 21626.657} C_VEL
LIN {X 0,Y 441.12,Z 370.014,A -85,B 0,C 180,E1 21622.938,E2 21622.938} C_VEL
LIN {X 0,Y 441.136,Z 370.025,A -85,B 0,C 180,E1 21619.317,E2 21619.317} C_VEL
LIN {X 0,Y 441.163,Z 370.007,A -85,B 0,C 180,E1 21615.593,E2 21615.593} C_VEL
LIN {X 0,Y 441.166,Z 370.021,A -85,B 0,C 180,E1 21611.896,E2 21611.896} C_VEL
LIN {X 0,Y 441.135,Z 370.006,A -85,B 0,C 180,E1 21608.203,E2 21608.203} C_VEL
LIN {X 0,Y 441.123,Z 370.032,A -85,B 0,C 180,E1 21604.544,E2 21604.544} C_VEL
LIN {X 0,Y 441.122,Z 370.001,A -85,B 0,C 180,E1 21600.774,E2 21600.774} C_VEL
LIN {X 0,Y 441.163,Z 370.031,A -85,B 0,C 180,E1 21597.267,E2 21597.267} C_VEL
LIN {X 0,Y 441.177,Z 369.99,A -85,B 0,C 180,E1 21593.488,E2 21593.488} C_VEL
LIN {X 0,Y 441.146,Z 370.033,A -85,B 0,C 180,E1 21589.812,E2 21589.812} C_VEL
LIN {X 0,Y 441.12,Z 369.999,A -85,B 0,C 180,E1 21586.227,E2 21586.227} C_VEL
LIN {X 0,Y 441.126,Z 370.034,A -85,B 0,C 180,E1 21582.45,E2 21582.45} C_VEL
LIN {X 0,Y 441.152,Z 369.998,A -85,B 0,C 180,E1 21578.873,E2 21578.873} C_VEL
LIN {X 0,Y 441.176,Z 370.034,A -85,B 0,C 180,E1 21575.207,E2 21575.207} C_VEL
LIN {X 0,Y 441.152,Z 370.002,A -85,B 0,C 180,E1 21571.426,E2 21571.426} C_VEL
LIN {X 0,Y 441.128,Z 370.027,A -85,B 0,C 180,E1 21567.811,E2 21567.811} C_VEL
LIN {X 0,Y 441.126,Z 370.035,A -85,B 0,C 180,E1 21564.013,E2 21564.013} C_VEL
LIN {X 0,Y 441.146,Z 370.036,A -85,B 0,C 180,E1 21560.407,E2 21560.407} C_VEL
LIN {X 0,Y 441.178,Z 370.033,A -85,B 0,C 180,E1 21556.805,E2 21556.805} C_VEL
LIN {X 0,Y 441.17,Z 370.267,A -85,B 0,C 180,E1 21553.403,E2 21553.403} C_VEL
LIN {X 0,Y 445.771,Z 385.008,A -85,B 0,C 180,E1 21550.238,E2 21550.238} C_VEL
LIN {X 0,Y 447.659,Z 391.164,A -85,B 0,C 180,E1 21549.061,E2 21549.061} C_VEL
LIN {X 0,Y 459.074,Z 412.595,A -85,B 0,C 180,E1 21547.498,E2 21547.498} C_VEL
LIN {X 0,Y 461.119,Z 419.25,A -85,B 0,C 180,E1 21547.178,E2 21547.178} C_VEL
LIN {X 0,Y 464.31,Z 432.479,A -85,B 0,C 180,E1 21546.633,E2 21546.633} C_VEL
LIN {X 0,Y 459.641,Z 648.48,A -85,B 0,C 180,E1 21542.999,E2 21542.999} C_VEL
LIN {X 0,Y 458.654,Z 668.877,A -85,B 0,C 180,E1 21542.49,E2 21542.49} C_VEL
LIN {X 0,Y 457.243,Z 688.444,A -85,B 0,C 180,E1 21541.765,E2 21541.765} C_VEL
LIN {X 0,Y 455.845,Z 704.873,A -85,B 0,C 180,E1 21540.986,E2 21540.986} C_VEL
LIN {X 0,Y 454.087,Z 723.201,A -85,B 0,C 180,E1 21539.918,E2 21539.918} C_VEL
LIN {X 0,Y 452.049,Z 741.549,A -85,B 0,C 180,E1 21538.582,E2 21538.582} C_VEL
LIN {X 0,Y 450.295,Z 756.486,A -85,B 0,C 180,E1 21537.291,E2 21537.291} C_VEL
LIN {X 0,Y 448.334,Z 772.887,A -85,B 0,C 180,E1 21535.635,E2 21535.635} C_VEL
LIN {X 0,Y 446.398,Z 788.214,A -85,B 0,C 180,E1 21533.776,E2 21533.776} C_VEL
LIN {X 0,Y 444.899,Z 800.543,A -85,B 0,C 180,E1 21532.043,E2 21532.043} C_VEL
LIN {X 0,Y 443.4,Z 813.799,A -85,B 0,C 180,E1 21529.888,E2 21529.888} C_VEL
LIN {X 0,Y 442.174,Z 825.288,A -85,B 0,C 180,E1 21527.638,E2 21527.638} C_VEL
LIN {X 0,Y 441.368,Z 834.036,A -85,B 0,C 180,E1 21525.639,E2 21525.639} C_VEL
LIN {X 0,Y 440.694,Z 842.915,A -85,B 0,C 180,E1 21523.247,E2 21523.247} C_VEL
LIN {X 0,Y 440.261,Z 850.312,A -85,B 0,C 180,E1 21520.732,E2 21520.732} C_VEL
LIN {X 0,Y 440.054,Z 855.53,A -85,B 0,C 180,E1 21518.493,E2 21518.493} C_VEL
LIN {X 0,Y 439.952,Z 859.501,A -85,B 0,C 180,E1 21516.263,E2 21516.263} C_VEL
LIN {X 0,Y 439.92,Z 862.728,A -85,B 0,C 180,E1 21513.518,E2 21513.518} C_VEL
LIN {X 0,Y 439.918,Z 863.987,A -85,B 0,C 180,E1 21511.172,E2 21511.172} C_VEL
LIN {X 0,Y 439.92,Z 864.046,A -85,B 0,C 180,E1 21509.088,E2 21509.088} C_VEL
LIN {X 0,Y 439.921,Z 862.994,A -85,B 0,C 180,E1 21506.873,E2 21506.873} C_VEL
LIN {X 0,Y 439.943,Z 860.329,A -85,B 0,C 180,E1 21504.261,E2 21504.261} C_VEL
LIN {X 0,Y 440.031,Z 856.072,A -85,B 0,C 180,E1 21501.77,E2 21501.77} C_VEL
LIN {X 0,Y 440.218,Z 851.092,A -85,B 0,C 180,E1 21499.575,E2 21499.575} C_VEL
LIN {X 0,Y 440.579,Z 844.586,A -85,B 0,C 180,E1 21497.283,E2 21497.283} C_VEL
LIN {X 0,Y 441.28,Z 835.123,A -85,B 0,C 180,E1 21494.628,E2 21494.628} C_VEL
LIN {X 0,Y 442.052,Z 826.53,A -85,B 0,C 180,E1 21492.629,E2 21492.629} C_VEL
LIN {X 0,Y 443.083,Z 816.449,A -85,B 0,C 180,E1 21490.611,E2 21490.611} C_VEL
LIN {X 0,Y 444.7,Z 802.302,A -85,B 0,C 180,E1 21488.22,E2 21488.22} C_VEL
LIN {X 0,Y 446.22,Z 789.672,A -85,B 0,C 180,E1 21486.418,E2 21486.418} C_VEL
LIN {X 0,Y 447.869,Z 776.311,A -85,B 0,C 180,E1 21484.761,E2 21484.761} C_VEL
LIN {X 0,Y 450.052,Z 758.625,A -85,B 0,C 180,E1 21482.908,E2 21482.908} C_VEL
LIN {X 0,Y 451.797,Z 743.659,A -85,B 0,C 180,E1 21481.589,E2 21481.589} C_VEL
LIN {X 0,Y 453.563,Z 727.981,A -85,B 0,C 180,E1 21480.411,E2 21480.411} C_VEL
LIN {X 0,Y 455.58,Z 707.926,A -85,B 0,C 180,E1 21479.173,E2 21479.173} C_VEL
LIN {X 0,Y 457.056,Z 690.676,A -85,B 0,C 180,E1 21478.331,E2 21478.331} C_VEL
LIN {X 0,Y 458.314,Z 673.745,A -85,B 0,C 180,E1 21477.678,E2 21477.678} C_VEL
LIN {X 0,Y 459.492,Z 652.797,A -85,B 0,C 180,E1 21477.086,E2 21477.086} C_VEL
LIN {X 0,Y 460.501,Z 612.198,A -85,B 0,C 180,E1 21476.373,E2 21476.373} C_VEL
LIN {X 0,Y 464.235,Z 431.351,A -85,B 0,C 180,E1 21473.339,E2 21473.339} C_VEL
LIN {X 0,Y 459.247,Z 412.946,A -85,B 0,C 180,E1 21472.525,E2 21472.525} C_VEL
LIN {X 0,Y 449.661,Z 395.012,A -85,B 0,C 180,E1 21471.232,E2 21471.232} C_VEL
LIN {X 0,Y 447.505,Z 390.733,A -85,B 0,C 180,E1 21470.887,E2 21470.887} C_VEL
LIN {X 0,Y 443.184,Z 376.751,A -85,B 0,C 180,E1 21468.024,E2 21468.024} C_VEL
LIN {X 0,Y 441.146,Z 370.123,A -85,B 0,C 180,E1 21466.545,E2 21466.545} C_VEL
LIN {X 0,Y 441.159,Z 370.03,A -85,B 0,C 180,E1 21462.842,E2 21462.842} C_VEL
LIN {X 0,Y 441.189,Z 370.023,A -85,B 0,C 180,E1 21459.056,E2 21459.056} C_VEL
LIN {X 0,Y 441.161,Z 370.034,A -85,B 0,C 180,E1 21455.31,E2 21455.31} C_VEL
LIN {X 0,Y 441.131,Z 370.031,A -85,B 0,C 180,E1 21451.729,E2 21451.729} C_VEL
LIN {X 0,Y 441.123,Z 370.002,A -85,B 0,C 180,E1 21447.986,E2 21447.986} C_VEL
LIN {X 0,Y 441.141,Z 370.033,A -85,B 0,C 180,E1 21444.34,E2 21444.34} C_VEL
LIN {X 0,Y 441.175,Z 369.998,A -85,B 0,C 180,E1 21440.709,E2 21440.709} C_VEL
LIN {X 0,Y 441.162,Z 370.03,A -85,B 0,C 180,E1 21436.981,E2 21436.981} C_VEL
LIN {X 0,Y 441.123,Z 370.001,A -85,B 0,C 180,E1 21433.505,E2 21433.505} C_VEL
LIN {X 0,Y 441.126,Z 370.033,A -85,B 0,C 180,E1 21429.793,E2 21429.793} C_VEL
LIN {X 0,Y 441.14,Z 369.995,A -85,B 0,C 180,E1 21426.12,E2 21426.12} C_VEL
LIN {X 0,Y 441.175,Z 370.033,A -85,B 0,C 180,E1 21422.473,E2 21422.473} C_VEL
LIN {X 0,Y 441.14,Z 369.995,A -85,B 0,C 180,E1 21418.837,E2 21418.837} C_VEL
LIN {X 0,Y 441.126,Z 370.031,A -85,B 0,C 180,E1 21415.195,E2 21415.195} C_VEL
LIN {X 0,Y 441.12,Z 370.003,A -85,B 0,C 180,E1 21411.403,E2 21411.403} C_VEL
LIN {X 0,Y 441.134,Z 370.034,A -85,B 0,C 180,E1 21407.65,E2 21407.65} C_VEL
LIN {X 0,Y 441.17,Z 370,A -85,B 0,C 180,E1 21404.091,E2 21404.091} C_VEL
LIN {X 0,Y 441.17,Z 370.025,A -85,B 0,C 180,E1 21400.271,E2 21400.271} C_VEL
LIN {X 0,Y 441.135,Z 370.006,A -85,B 0,C 180,E1 21396.625,E2 21396.625} C_VEL
LIN {X 0,Y 441.124,Z 370.035,A -85,B 0,C 180,E1 21392.906,E2 21392.906} C_VEL
LIN {X 0,Y 441.126,Z 370.035,A -85,B 0,C 180,E1 21389.195,E2 21389.195} C_VEL
LIN {X 0,Y 441.152,Z 370.035,A -85,B 0,C 180,E1 21385.586,E2 21385.586} C_VEL
LIN {X 0,Y 441.179,Z 370.033,A -85,B 0,C 180,E1 21381.789,E2 21381.789} C_VEL
LIN {X 0,Y 441.157,Z 370.035,A -85,B 0,C 180,E1 21378.052,E2 21378.052} C_VEL
LIN {X 0,Y 441.126,Z 370.036,A -85,B 0,C 180,E1 21374.453,E2 21374.453} C_VEL
LIN {X 0,Y 441.12,Z 370.035,A -85,B 0,C 180,E1 21370.751,E2 21370.751} C_VEL
LIN {X 0,Y 441.136,Z 370.034,A -85,B 0,C 180,E1 21367.092,E2 21367.092} C_VEL
LIN {X 0,Y 441.171,Z 370.031,A -85,B 0,C 180,E1 21363.416,E2 21363.416} C_VEL
LIN {X 0,Y 441.171,Z 370.033,A -85,B 0,C 180,E1 21359.607,E2 21359.607} C_VEL
LIN {X 0,Y 441.14,Z 370.037,A -85,B 0,C 180,E1 21355.888,E2 21355.888} C_VEL
LIN {X 0,Y 441.121,Z 370.036,A -85,B 0,C 180,E1 21352.242,E2 21352.242} C_VEL
LIN {X 0,Y 441.121,Z 370.036,A -85,B 0,C 180,E1 21348.501,E2 21348.501} C_VEL
LIN {X 0,Y 441.141,Z 370.037,A -85,B 0,C 180,E1 21344.839,E2 21344.839} C_VEL
LIN {X 0,Y 441.167,Z 370.033,A -85,B 0,C 180,E1 21341.134,E2 21341.134} C_VEL
LIN {X 0,Y 441.15,Z 370.033,A -85,B 0,C 180,E1 21337.423,E2 21337.423} C_VEL
LIN {X 0,Y 441.124,Z 370.038,A -85,B 0,C 180,E1 21336.418,E2 21336.418} C_VEL
LIN {X 0,Y 440.106,Z 370.164,A -85,B 0,C 180,E1 21335.417,E2 21335.417} C_VEL
LIN {X 0,Y 433.603,Z 370.974,A -85,B 0,C 180,E1 21332.527,E2 21332.527} C_VEL
LIN {X 0,Y 433.179,Z 371.027,A -85,B 0,C 180,E1 21331.864,E2 21331.864} C_VEL
LIN {X 0,Y 433.178,Z 371.027,A -85,B 0,C 180,E1 21328.016,E2 21328.016} C_VEL
LIN {X 0,Y 433.189,Z 371.024,A -85,B 0,C 180,E1 21324.304,E2 21324.304} C_VEL
LIN {X 0,Y 433.224,Z 371.021,A -85,B 0,C 180,E1 21320.703,E2 21320.703} C_VEL
LIN {X 0,Y 433.232,Z 371.022,A -85,B 0,C 180,E1 21316.847,E2 21316.847} C_VEL
LIN {X 0,Y 433.196,Z 371.024,A -85,B 0,C 180,E1 21313.232,E2 21313.232} C_VEL
LIN {X 0,Y 433.181,Z 371.024,A -85,B 0,C 180,E1 21309.546,E2 21309.546} C_VEL
LIN {X 0,Y 433.182,Z 371.027,A -85,B 0,C 180,E1 21305.722,E2 21305.722} C_VEL
LIN {X 0,Y 433.198,Z 371.025,A -85,B 0,C 180,E1 21302.061,E2 21302.061} C_VEL
LIN {X 0,Y 433.231,Z 371.02,A -85,B 0,C 180,E1 21298.37,E2 21298.37} C_VEL
LIN {X 0,Y 433.229,Z 371.02,A -85,B 0,C 180,E1 21294.541,E2 21294.541} C_VEL
LIN {X 0,Y 433.204,Z 371.022,A -85,B 0,C 180,E1 21290.773,E2 21290.773} C_VEL
LIN {X 0,Y 433.184,Z 371.025,A -85,B 0,C 180,E1 21287.209,E2 21287.209} C_VEL
LIN {X 0,Y 433.183,Z 371.026,A -85,B 0,C 180,E1 21283.36,E2 21283.36} C_VEL
LIN {X 0,Y 433.203,Z 371.023,A -85,B 0,C 180,E1 21279.731,E2 21279.731} C_VEL
LIN {X 0,Y 433.232,Z 371.022,A -85,B 0,C 180,E1 21276.042,E2 21276.042} C_VEL
LIN {X 0,Y 433.23,Z 371.022,A -85,B 0,C 180,E1 21272.208,E2 21272.208} C_VEL
LIN {X 0,Y 433.2,Z 371.024,A -85,B 0,C 180,E1 21268.531,E2 21268.531} C_VEL
LIN {X 0,Y 433.182,Z 370.996,A -85,B 0,C 180,E1 21264.832,E2 21264.832} C_VEL
LIN {X 0,Y 433.184,Z 371.024,A -85,B 0,C 180,E1 21260.955,E2 21260.955} C_VEL
LIN {X 0,Y 433.197,Z 370.983,A -85,B 0,C 180,E1 21257.315,E2 21257.315} C_VEL
LIN {X 0,Y 433.232,Z 371.023,A -85,B 0,C 180,E1 21253.609,E2 21253.609} C_VEL
LIN {X 0,Y 433.229,Z 370.979,A -85,B 0,C 180,E1 21249.785,E2 21249.785} C_VEL
LIN {X 0,Y 433.195,Z 371.019,A -85,B 0,C 180,E1 21246.222,E2 21246.222} C_VEL
LIN {X 0,Y 433.18,Z 370.99,A -85,B 0,C 180,E1 21242.508,E2 21242.508} C_VEL
LIN {X 0,Y 433.186,Z 371.02,A -85,B 0,C 180,E1 21238.672,E2 21238.672} C_VEL
LIN {X 0,Y 433.199,Z 370.996,A -85,B 0,C 180,E1 21234.963,E2 21234.963} C_VEL
LIN {X 0,Y 433.238,Z 371.003,A -85,B 0,C 180,E1 21231.367,E2 21231.367} C_VEL
LIN {X 0,Y 433.219,Z 370.999,A -85,B 0,C 180,E1 21227.601,E2 21227.601} C_VEL
LIN {X 0,Y 433.189,Z 371.009,A -85,B 0,C 180,E1 21224.053,E2 21224.053} C_VEL
LIN {X 0,Y 433.186,Z 371.01,A -85,B 0,C 180,E1 21220.302,E2 21220.302} C_VEL
LIN {X 0,Y 433.199,Z 371.014,A -85,B 0,C 180,E1 21216.605,E2 21216.605} C_VEL
LIN {X 0,Y 433.234,Z 370.989,A -85,B 0,C 180,E1 21212.953,E2 21212.953} C_VEL
LIN {X 0,Y 433.24,Z 371.022,A -85,B 0,C 180,E1 21209.148,E2 21209.148} C_VEL
LIN {X 0,Y 433.209,Z 371.013,A -85,B 0,C 180,E1 21205.401,E2 21205.401} C_VEL
LIN {X 0,Y 433.191,Z 371.008,A -85,B 0,C 180,E1 21201.697,E2 21201.697} C_VEL
LIN {X 0,Y 433.188,Z 371.011,A -85,B 0,C 180,E1 21197.978,E2 21197.978} C_VEL
LIN {X 0,Y 433.212,Z 371.1,A -85,B 0,C 180,E1 21194.218,E2 21194.218} C_VEL
LIN {X 0,Y 437.433,Z 384.319,A -85,B 0,C 180,E1 21191.231,E2 21191.231} C_VEL
LIN {X 0,Y 439.409,Z 390.873,A -85,B 0,C 180,E1 21189.939,E2 21189.939} C_VEL
LIN {X 0,Y 450.989,Z 412.262,A -85,B 0,C 180,E1 21188.291,E2 21188.291} C_VEL
LIN {X 0,Y 454.096,Z 418.791,A -85,B 0,C 180,E1 21187.857,E2 21187.857} C_VEL
LIN {X 0,Y 457.846,Z 434.192,A -85,B 0,C 180,E1 21187.199,E2 21187.199} C_VEL
LIN {X 0,Y 452.92,Z 648.551,A -85,B 0,C 180,E1 21183.546,E2 21183.546} C_VEL
LIN {X 0,Y 451.846,Z 669.269,A -85,B 0,C 180,E1 21183.017,E2 21183.017} C_VEL
LIN {X 0,Y 450.406,Z 688.205,A -85,B 0,C 180,E1 21182.305,E2 21182.305} C_VEL
LIN {X 0,Y 448.996,Z 703.949,A -85,B 0,C 180,E1 21181.554,E2 21181.554} C_VEL
LIN {X 0,Y 447.163,Z 721.943,A -85,B 0,C 180,E1 21180.501,E2 21180.501} C_VEL
LIN {X 0,Y 444.954,Z 740.995,A -85,B 0,C 180,E1 21179.11,E2 21179.11} C_VEL
LIN {X 0,Y 443.071,Z 756.065,A -85,B 0,C 180,E1 21177.792,E2 21177.792} C_VEL
LIN {X 0,Y 441.11,Z 771.381,A -85,B 0,C 180,E1 21176.231,E2 21176.231} C_VEL
LIN {X 0,Y 438.958,Z 787.47,A -85,B 0,C 180,E1 21174.276,E2 21174.276} C_VEL
LIN {X 0,Y 437.292,Z 800.3,A -85,B 0,C 180,E1 21172.447,E2 21172.447} C_VEL
LIN {X 0,Y 435.694,Z 813.455,A -85,B 0,C 180,E1 21170.274,E2 21170.274} C_VEL
LIN {X 0,Y 434.36,Z 825.045,A -85,B 0,C 180,E1 21167.966,E2 21167.966} C_VEL
LIN {X 0,Y 433.466,Z 834.055,A -85,B 0,C 180,E1 21165.865,E2 21165.865} C_VEL
LIN {X 0,Y 432.728,Z 843.131,A -85,B 0,C 180,E1 21163.359,E2 21163.359} C_VEL
LIN {X 0,Y 432.27,Z 850.408,A -85,B 0,C 180,E1 21160.798,E2 21160.798} C_VEL
LIN {X 0,Y 432.061,Z 855.291,A -85,B 0,C 180,E1 21158.651,E2 21158.651} C_VEL
LIN {X 0,Y 431.955,Z 859.263,A -85,B 0,C 180,E1 21156.379,E2 21156.379} C_VEL
LIN {X 0,Y 431.923,Z 862.491,A -85,B 0,C 180,E1 21153.583,E2 21153.583} C_VEL
LIN {X 0,Y 431.921,Z 863.751,A -85,B 0,C 180,E1 21151.194,E2 21151.194} C_VEL
LIN {X 0,Y 431.924,Z 863.81,A -85,B 0,C 180,E1 21149.072,E2 21149.072} C_VEL
LIN {X 0,Y 431.923,Z 862.758,A -85,B 0,C 180,E1 21146.815,E2 21146.815} C_VEL
LIN {X 0,Y 431.946,Z 860.091,A -85,B 0,C 180,E1 21144.154,E2 21144.154} C_VEL
LIN {X 0,Y 432.046,Z 855.833,A -85,B 0,C 180,E1 21141.617,E2 21141.617} C_VEL
LIN {X 0,Y 432.234,Z 851.072,A -85,B 0,C 180,E1 21139.468,E2 21139.468} C_VEL
LIN {X 0,Y 432.606,Z 844.746,A -85,B 0,C 180,E1 21137.181,E2 21137.181} C_VEL
LIN {X 0,Y 433.348,Z 835.425,A -85,B 0,C 180,E1 21134.476,E2 21134.476} C_VEL
LIN {X 0,Y 434.229,Z 826.288,A -85,B 0,C 180,E1 21132.306,E2 21132.306} C_VEL
LIN {X 0,Y 435.33,Z 816.291,A -85,B 0,C 180,E1 21130.268,E2 21130.268} C_VEL
LIN {X 0,Y 436.994,Z 802.744,A -85,B 0,C 180,E1 21127.924,E2 21127.924} C_VEL
LIN {X 0,Y 438.695,Z 789.475,A -85,B 0,C 180,E1 21125.995,E2 21125.995} C_VEL
LIN {X 0,Y 440.469,Z 776.069,A -85,B 0,C 180,E1 21124.307,E2 21124.307} C_VEL
LIN {X 0,Y 442.784,Z 758.383,A -85,B 0,C 180,E1 21122.426,E2 21122.426} C_VEL
LIN {X 0,Y 444.646,Z 743.419,A -85,B 0,C 180,E1 21121.089,E2 21121.089} C_VEL
LIN {X 0,Y 446.514,Z 727.741,A -85,B 0,C 180,E1 21119.896,E2 21119.896} C_VEL
LIN {X 0,Y 448.657,Z 707.562,A -85,B 0,C 180,E1 21118.637,E2 21118.637} C_VEL
LIN {X 0,Y 450.211,Z 690.438,A -85,B 0,C 180,E1 21117.792,E2 21117.792} C_VEL
LIN {X 0,Y 451.526,Z 673.622,A -85,B 0,C 180,E1 21117.136,E2 21117.136} C_VEL
LIN {X 0,Y 452.763,Z 652.856,A -85,B 0,C 180,E1 21116.54,E2 21116.54} C_VEL
LIN {X 0,Y 453.81,Z 613.363,A -85,B 0,C 180,E1 21115.835,E2 21115.835} C_VEL
LIN {X 0,Y 457.748,Z 433.077,A -85,B 0,C 180,E1 21112.77,E2 21112.77} C_VEL
LIN {X 0,Y 453.367,Z 416.797,A -85,B 0,C 180,E1 21112.033,E2 21112.033} C_VEL
LIN {X 0,Y 443.722,Z 398.797,A -85,B 0,C 180,E1 21110.695,E2 21110.695} C_VEL
LIN {X 0,Y 439.212,Z 390.386,A -85,B 0,C 180,E1 21110.003,E2 21110.003} C_VEL
LIN {X 0,Y 435.007,Z 376.564,A -85,B 0,C 180,E1 21107.074,E2 21107.074} C_VEL
LIN {X 0,Y 433.211,Z 371.085,A -85,B 0,C 180,E1 21105.767,E2 21105.767} C_VEL
LIN {X 0,Y 433.188,Z 371.011,A -85,B 0,C 180,E1 21102.022,E2 21102.022} C_VEL
LIN {X 0,Y 433.188,Z 371.007,A -85,B 0,C 180,E1 21098.217,E2 21098.217} C_VEL
LIN {X 0,Y 433.204,Z 371.013,A -85,B 0,C 180,E1 21094.518,E2 21094.518} C_VEL
LIN {X 0,Y 433.238,Z 371.021,A -85,B 0,C 180,E1 21090.825,E2 21090.825} C_VEL
LIN {X 0,Y 433.235,Z 370.989,A -85,B 0,C 180,E1 21087.024,E2 21087.024} C_VEL
LIN {X 0,Y 433.209,Z 371.009,A -85,B 0,C 180,E1 21083.25,E2 21083.25} C_VEL
LIN {X 0,Y 433.189,Z 371.012,A -85,B 0,C 180,E1 21079.558,E2 21079.558} C_VEL
LIN {X 0,Y 433.185,Z 371.006,A -85,B 0,C 180,E1 21075.746,E2 21075.746} C_VEL
LIN {X 0,Y 433.193,Z 371.012,A -85,B 0,C 180,E1 21071.994,E2 21071.994} C_VEL
LIN {X 0,Y 433.222,Z 371.001,A -85,B 0,C 180,E1 21068.366,E2 21068.366} C_VEL
LIN {X 0,Y 433.229,Z 370.997,A -85,B 0,C 180,E1 21064.639,E2 21064.639} C_VEL
LIN {X 0,Y 433.204,Z 371.013,A -85,B 0,C 180,E1 21060.931,E2 21060.931} C_VEL
LIN {X 0,Y 433.183,Z 370.995,A -85,B 0,C 180,E1 21057.228,E2 21057.228} C_VEL
LIN {X 0,Y 433.184,Z 371.019,A -85,B 0,C 180,E1 21053.512,E2 21053.512} C_VEL
LIN {X 0,Y 433.203,Z 370.985,A -85,B 0,C 180,E1 21049.904,E2 21049.904} C_VEL
LIN {X 0,Y 433.234,Z 371.018,A -85,B 0,C 180,E1 21046.119,E2 21046.119} C_VEL
LIN {X 0,Y 433.219,Z 370.982,A -85,B 0,C 180,E1 21042.395,E2 21042.395} C_VEL
LIN {X 0,Y 433.192,Z 371.023,A -85,B 0,C 180,E1 21038.762,E2 21038.762} C_VEL
LIN {X 0,Y 433.181,Z 370.999,A -85,B 0,C 180,E1 21035.022,E2 21035.022} C_VEL
LIN {X 0,Y 433.19,Z 371.024,A -85,B 0,C 180,E1 21031.29,E2 21031.29} C_VEL
LIN {X 0,Y 433.23,Z 371.022,A -85,B 0,C 180,E1 21027.792,E2 21027.792} C_VEL
LIN {X 0,Y 433.232,Z 371.022,A -85,B 0,C 180,E1 21023.958,E2 21023.958} C_VEL
LIN {X 0,Y 433.207,Z 371.023,A -85,B 0,C 180,E1 21020.224,E2 21020.224} C_VEL
LIN {X 0,Y 433.184,Z 371.025,A -85,B 0,C 180,E1 21016.553,E2 21016.553} C_VEL
LIN {X 0,Y 433.183,Z 371.025,A -85,B 0,C 180,E1 21012.733,E2 21012.733} C_VEL
LIN {X 0,Y 433.189,Z 371.023,A -85,B 0,C 180,E1 21008.951,E2 21008.951} C_VEL
LIN {X 0,Y 433.212,Z 371.022,A -85,B 0,C 180,E1 21005.239,E2 21005.239} C_VEL
LIN {X 0,Y 433.235,Z 371.021,A -85,B 0,C 180,E1 21001.437,E2 21001.437} C_VEL
LIN {X 0,Y 433.23,Z 371.023,A -85,B 0,C 180,E1 20997.616,E2 20997.616} C_VEL
LIN {X 0,Y 433.203,Z 371.023,A -85,B 0,C 180,E1 20993.822,E2 20993.822} C_VEL
LIN {X 0,Y 433.179,Z 371.024,A -85,B 0,C 180,E1 20990.256,E2 20990.256} C_VEL
LIN {X 0,Y 433.184,Z 371.027,A -85,B 0,C 180,E1 20986.493,E2 20986.493} C_VEL
LIN {X 0,Y 433.214,Z 371.024,A -85,B 0,C 180,E1 20982.936,E2 20982.936} C_VEL
LIN {X 0,Y 433.231,Z 371.02,A -85,B 0,C 180,E1 20979.163,E2 20979.163} C_VEL
LIN {X 0,Y 433.208,Z 371.022,A -85,B 0,C 180,E1 20975.43,E2 20975.43} C_VEL
LIN {X 0,Y 433.179,Z 371.027,A -85,B 0,C 180,E1 20971.864,E2 20971.864} C_VEL
LIN {X 0,Y 432.194,Z 371.152,A -85,B 0,C 180,E1 20970.845,E2 20970.845} C_VEL
LIN {X 0,Y 425.761,Z 371.951,A -85,B 0,C 180,E1 20967.974,E2 20967.974} C_VEL
LIN {X 0,Y 425.272,Z 372.011,A -85,B 0,C 180,E1 20967.224,E2 20967.224} C_VEL
LIN {X 0,Y 425.249,Z 372.016,A -85,B 0,C 180,E1 20963.52,E2 20963.52} C_VEL
LIN {X 0,Y 425.24,Z 372.015,A -85,B 0,C 180,E1 20959.843,E2 20959.843} C_VEL
LIN {X 0,Y 425.242,Z 372.014,A -85,B 0,C 180,E1 20955.985,E2 20955.985} C_VEL
LIN {X 0,Y 425.27,Z 372.013,A -85,B 0,C 180,E1 20952.345,E2 20952.345} C_VEL
LIN {X 0,Y 425.295,Z 372.009,A -85,B 0,C 180,E1 20948.563,E2 20948.563} C_VEL
LIN {X 0,Y 425.29,Z 372.008,A -85,B 0,C 180,E1 20944.668,E2 20944.668} C_VEL
LIN {X 0,Y 425.27,Z 372.011,A -85,B 0,C 180,E1 20940.878,E2 20940.878} C_VEL
LIN {X 0,Y 425.246,Z 372.015,A -85,B 0,C 180,E1 20937.264,E2 20937.264} C_VEL
LIN {X 0,Y 425.244,Z 372.015,A -85,B 0,C 180,E1 20933.498,E2 20933.498} C_VEL
LIN {X 0,Y 425.252,Z 372.012,A -85,B 0,C 180,E1 20929.717,E2 20929.717} C_VEL
LIN {X 0,Y 425.275,Z 372.01,A -85,B 0,C 180,E1 20925.995,E2 20925.995} C_VEL
LIN {X 0,Y 425.297,Z 372.009,A -85,B 0,C 180,E1 20922.223,E2 20922.223} C_VEL
LIN {X 0,Y 425.274,Z 372.011,A -85,B 0,C 180,E1 20918.474,E2 20918.474} C_VEL
LIN {X 0,Y 425.249,Z 372.015,A -85,B 0,C 180,E1 20914.834,E2 20914.834} C_VEL
LIN {X 0,Y 425.246,Z 372.013,A -85,B 0,C 180,E1 20911.14,E2 20911.14} C_VEL
LIN {X 0,Y 425.259,Z 372.013,A -85,B 0,C 180,E1 20907.432,E2 20907.432} C_VEL
LIN {X 0,Y 425.28,Z 371.975,A -85,B 0,C 180,E1 20903.697,E2 20903.697} C_VEL
LIN {X 0,Y 425.295,Z 372.005,A -85,B 0,C 180,E1 20899.923,E2 20899.923} C_VEL
LIN {X 0,Y 425.274,Z 371.974,A -85,B 0,C 180,E1 20896.1,E2 20896.1} C_VEL
LIN {X 0,Y 425.249,Z 372.012,A -85,B 0,C 180,E1 20892.486,E2 20892.486} C_VEL
LIN {X 0,Y 425.242,Z 371.976,A -85,B 0,C 180,E1 20888.648,E2 20888.648} C_VEL
LIN {X 0,Y 425.251,Z 372.009,A -85,B 0,C 180,E1 20884.849,E2 20884.849} C_VEL
LIN {X 0,Y 425.255,Z 371.97,A -85,B 0,C 180,E1 20881.072,E2 20881.072} C_VEL
LIN {X 0,Y 425.294,Z 372.01,A -85,B 0,C 180,E1 20877.434,E2 20877.434} C_VEL
LIN {X 0,Y 425.295,Z 371.964,A -85,B 0,C 180,E1 20873.515,E2 20873.515} C_VEL
LIN {X 0,Y 425.276,Z 372.011,A -85,B 0,C 180,E1 20869.702,E2 20869.702} C_VEL
LIN {X 0,Y 425.249,Z 371.971,A -85,B 0,C 180,E1 20865.98,E2 20865.98} C_VEL
LIN {X 0,Y 425.246,Z 372.013,A -85,B 0,C 180,E1 20862.197,E2 20862.197} C_VEL
LIN {X 0,Y 425.246,Z 371.976,A -85,B 0,C 180,E1 20858.332,E2 20858.332} C_VEL
LIN {X 0,Y 425.268,Z 372.008,A -85,B 0,C 180,E1 20854.661,E2 20854.661} C_VEL
LIN {X 0,Y 425.29,Z 371.984,A -85,B 0,C 180,E1 20850.875,E2 20850.875} C_VEL
LIN {X 0,Y 425.294,Z 371.988,A -85,B 0,C 180,E1 20847.102,E2 20847.102} C_VEL
LIN {X 0,Y 425.275,Z 372,A -85,B 0,C 180,E1 20843.292,E2 20843.292} C_VEL
LIN {X 0,Y 425.253,Z 372.009,A -85,B 0,C 180,E1 20839.62,E2 20839.62} C_VEL
LIN {X 0,Y 425.25,Z 372.004,A -85,B 0,C 180,E1 20835.816,E2 20835.816} C_VEL
LIN {X 0,Y 425.338,Z 372.305,A -85,B 0,C 180,E1 20834.917,E2 20834.917} C_VEL
LIN {X 0,Y 429.811,Z 386.383,A -85,B 0,C 180,E1 20831.688,E2 20831.688} C_VEL
LIN {X 0,Y 431.146,Z 390.518,A -85,B 0,C 180,E1 20830.865,E2 20830.865} C_VEL
LIN {X 0,Y 442.993,Z 411.939,A -85,B 0,C 180,E1 20829.113,E2 20829.113} C_VEL
LIN {X 0,Y 448.196,Z 422.471,A -85,B 0,C 180,E1 20828.368,E2 20828.368} C_VEL
LIN {X 0,Y 451.424,Z 436.081,A -85,B 0,C 180,E1 20827.778,E2 20827.778} C_VEL
LIN {X 0,Y 446.238,Z 648.725,A -85,B 0,C 180,E1 20824.107,E2 20824.107} C_VEL
LIN {X 0,Y 445.075,Z 669.605,A -85,B 0,C 180,E1 20823.561,E2 20823.561} C_VEL
LIN {X 0,Y 443.626,Z 687.77,A -85,B 0,C 180,E1 20822.871,E2 20822.871} C_VEL
LIN {X 0,Y 442.126,Z 703.71,A -85,B 0,C 180,E1 20822.102,E2 20822.102} C_VEL
LIN {X 0,Y 440.261,Z 721.047,A -85,B 0,C 180,E1 20821.079,E2 20821.079} C_VEL
LIN {X 0,Y 437.965,Z 739.946,A -85,B 0,C 180,E1 20819.695,E2 20819.695} C_VEL
LIN {X 0,Y 435.935,Z 755.29,A -85,B 0,C 180,E1 20818.344,E2 20818.344} C_VEL
LIN {X 0,Y 433.85,Z 770.507,A -85,B 0,C 180,E1 20816.778,E2 20816.778} C_VEL
LIN {X 0,Y 431.561,Z 786.726,A -85,B 0,C 180,E1 20814.793,E2 20814.793} C_VEL
LIN {X 0,Y 429.829,Z 799.164,A -85,B 0,C 180,E1 20813.003,E2 20813.003} C_VEL
LIN {X 0,Y 428.272,Z 810.836,A -85,B 0,C 180,E1 20811.071,E2 20811.071} C_VEL
LIN {X 0,Y 426.703,Z 823.56,A -85,B 0,C 180,E1 20808.582,E2 20808.582} C_VEL
LIN {X 0,Y 425.672,Z 833.009,A -85,B 0,C 180,E1 20806.371,E2 20806.371} C_VEL
LIN {X 0,Y 424.941,Z 841.021,A -85,B 0,C 180,E1 20804.164,E2 20804.164} C_VEL
LIN {X 0,Y 424.335,Z 849.497,A -85,B 0,C 180,E1 20801.278,E2 20801.278} C_VEL
LIN {X 0,Y 424.083,Z 854.844,A -85,B 0,C 180,E1 20798.92,E2 20798.92} C_VEL
LIN {X 0,Y 423.963,Z 858.816,A -85,B 0,C 180,E1 20796.636,E2 20796.636} C_VEL
LIN {X 0,Y 423.925,Z 862.103,A -85,B 0,C 180,E1 20793.881,E2 20793.881} C_VEL
LIN {X 0,Y 423.924,Z 863.514,A -85,B 0,C 180,E1 20791.216,E2 20791.216} C_VEL
LIN {X 0,Y 423.927,Z 863.574,A -85,B 0,C 180,E1 20789.054,E2 20789.054} C_VEL
LIN {X 0,Y 423.925,Z 862.521,A -85,B 0,C 180,E1 20786.755,E2 20786.755} C_VEL
LIN {X 0,Y 423.948,Z 859.854,A -85,B 0,C 180,E1 20784.044,E2 20784.044} C_VEL
LIN {X 0,Y 424.056,Z 855.595,A -85,B 0,C 180,E1 20781.458,E2 20781.458} C_VEL
LIN {X 0,Y 424.262,Z 850.838,A -85,B 0,C 180,E1 20779.27,E2 20779.27} C_VEL
LIN {X 0,Y 424.665,Z 844.506,A -85,B 0,C 180,E1 20776.937,E2 20776.937} C_VEL
LIN {X 0,Y 425.468,Z 835.183,A -85,B 0,C 180,E1 20774.181,E2 20774.181} C_VEL
LIN {X 0,Y 426.418,Z 826.045,A -85,B 0,C 180,E1 20771.971,E2 20771.971} C_VEL
LIN {X 0,Y 427.606,Z 816.048,A -85,B 0,C 180,E1 20769.897,E2 20769.897} C_VEL
LIN {X 0,Y 429.357,Z 802.737,A -85,B 0,C 180,E1 20767.549,E2 20767.549} C_VEL
LIN {X 0,Y 431.133,Z 789.734,A -85,B 0,C 180,E1 20765.62,E2 20765.62} C_VEL
LIN {X 0,Y 432.967,Z 776.705,A -85,B 0,C 180,E1 20763.943,E2 20763.943} C_VEL
LIN {X 0,Y 435.278,Z 760.352,A -85,B 0,C 180,E1 20762.139,E2 20762.139} C_VEL
LIN {X 0,Y 437.427,Z 743.986,A -85,B 0,C 180,E1 20760.641,E2 20760.641} C_VEL
LIN {X 0,Y 439.273,Z 729.346,A -85,B 0,C 180,E1 20759.498,E2 20759.498} C_VEL
LIN {X 0,Y 441.401,Z 711.06,A -85,B 0,C 180,E1 20758.297,E2 20758.297} C_VEL
LIN {X 0,Y 443.275,Z 691.686,A -85,B 0,C 180,E1 20757.302,E2 20757.302} C_VEL
LIN {X 0,Y 444.673,Z 674.873,A -85,B 0,C 180,E1 20756.626,E2 20756.626} C_VEL
LIN {X 0,Y 445.88,Z 656.573,A -85,B 0,C 180,E1 20756.07,E2 20756.07} C_VEL
LIN {X 0,Y 446.827,Z 628.929,A -85,B 0,C 180,E1 20755.527,E2 20755.527} C_VEL
LIN {X 0,Y 451.345,Z 434.944,A -85,B 0,C 180,E1 20752.192,E2 20752.192} C_VEL
LIN {X 0,Y 447.587,Z 420.803,A -85,B 0,C 180,E1 20751.538,E2 20751.538} C_VEL
LIN {X 0,Y 436.305,Z 399.683,A -85,B 0,C 180,E1 20749.918,E2 20749.918} C_VEL
LIN {X 0,Y 430.95,Z 390.001,A -85,B 0,C 180,E1 20749.072,E2 20749.072} C_VEL
LIN {X 0,Y 426.783,Z 376.996,A -85,B 0,C 180,E1 20746.189,E2 20746.189} C_VEL
LIN {X 0,Y 425.301,Z 372.102,A -85,B 0,C 180,E1 20745.002,E2 20745.002} C_VEL
LIN {X 0,Y 425.305,Z 371.992,A -85,B 0,C 180,E1 20741.171,E2 20741.171} C_VEL
LIN {X 0,Y 425.278,Z 371.992,A -85,B 0,C 180,E1 20737.379,E2 20737.379} C_VEL
LIN {X 0,Y 425.254,Z 371.992,A -85,B 0,C 180,E1 20733.664,E2 20733.664} C_VEL
LIN {X 0,Y 425.249,Z 372.009,A -85,B 0,C 180,E1 20729.903,E2 20729.903} C_VEL
LIN {X 0,Y 425.252,Z 372.002,A -85,B 0,C 180,E1 20726.086,E2 20726.086} C_VEL
LIN {X 0,Y 425.268,Z 371.981,A -85,B 0,C 180,E1 20722.393,E2 20722.393} C_VEL
LIN {X 0,Y 425.295,Z 372.004,A -85,B 0,C 180,E1 20718.652,E2 20718.652} C_VEL
LIN {X 0,Y 425.307,Z 371.966,A -85,B 0,C 180,E1 20714.713,E2 20714.713} C_VEL
LIN {X 0,Y 425.286,Z 372.007,A -85,B 0,C 180,E1 20710.846,E2 20710.846} C_VEL
LIN {X 0,Y 425.253,Z 371.974,A -85,B 0,C 180,E1 20707.164,E2 20707.164} C_VEL
LIN {X 0,Y 425.246,Z 372.009,A -85,B 0,C 180,E1 20703.375,E2 20703.375} C_VEL
LIN {X 0,Y 425.243,Z 371.98,A -85,B 0,C 180,E1 20699.602,E2 20699.602} C_VEL
LIN {X 0,Y 425.258,Z 372.004,A -85,B 0,C 180,E1 20695.826,E2 20695.826} C_VEL
LIN {X 0,Y 425.289,Z 371.982,A -85,B 0,C 180,E1 20692.169,E2 20692.169} C_VEL
LIN {X 0,Y 425.292,Z 371.993,A -85,B 0,C 180,E1 20688.342,E2 20688.342} C_VEL
LIN {X 0,Y 425.267,Z 371.988,A -85,B 0,C 180,E1 20684.6,E2 20684.6} C_VEL
LIN {X 0,Y 425.247,Z 372.003,A -85,B 0,C 180,E1 20680.932,E2 20680.932} C_VEL
LIN {X 0,Y 425.243,Z 371.99,A -85,B 0,C 180,E1 20677.171,E2 20677.171} C_VEL
LIN {X 0,Y 425.258,Z 372.011,A -85,B 0,C 180,E1 20673.475,E2 20673.475} C_VEL
LIN {X 0,Y 425.291,Z 372.011,A -85,B 0,C 180,E1 20669.803,E2 20669.803} C_VEL
LIN {X 0,Y 425.292,Z 372.012,A -85,B 0,C 180,E1 20665.986,E2 20665.986} C_VEL
LIN {X 0,Y 425.275,Z 372.011,A -85,B 0,C 180,E1 20662.158,E2 20662.158} C_VEL
LIN {X 0,Y 425.248,Z 372.014,A -85,B 0,C 180,E1 20658.479,E2 20658.479} C_VEL
LIN {X 0,Y 425.244,Z 372.015,A -85,B 0,C 180,E1 20654.669,E2 20654.669} C_VEL
LIN {X 0,Y 425.244,Z 372.013,A -85,B 0,C 180,E1 20650.804,E2 20650.804} C_VEL
LIN {X 0,Y 425.264,Z 372.011,A -85,B 0,C 180,E1 20647.167,E2 20647.167} C_VEL
LIN {X 0,Y 425.288,Z 372.009,A -85,B 0,C 180,E1 20643.375,E2 20643.375} C_VEL
LIN {X 0,Y 425.296,Z 372.01,A -85,B 0,C 180,E1 20639.577,E2 20639.577} C_VEL
LIN {X 0,Y 425.27,Z 372.013,A -85,B 0,C 180,E1 20635.782,E2 20635.782} C_VEL
LIN {X 0,Y 425.248,Z 372.013,A -85,B 0,C 180,E1 20632.098,E2 20632.098} C_VEL
LIN {X 0,Y 425.242,Z 372.015,A -85,B 0,C 180,E1 20628.364,E2 20628.364} C_VEL
LIN {X 0,Y 425.248,Z 372.016,A -85,B 0,C 180,E1 20624.571,E2 20624.571} C_VEL
LIN {X 0,Y 425.269,Z 372.011,A -85,B 0,C 180,E1 20620.841,E2 20620.841} C_VEL
LIN {X 0,Y 425.294,Z 372.008,A -85,B 0,C 180,E1 20617.022,E2 20617.022} C_VEL
LIN {X 0,Y 425.286,Z 372.012,A -85,B 0,C 180,E1 20613.1,E2 20613.1} C_VEL
LIN {X 0,Y 425.268,Z 372.011,A -85,B 0,C 180,E1 20609.326,E2 20609.326} C_VEL
LIN {X 0,Y 425.272,Z 372.011,A -85,B 0,C 180,E1 20607.224,E2 20607.224} C_VEL
LIN {X 0,Y 424.348,Z 372.129,A -85,B 0,C 180,E1 20606.187,E2 20606.187} C_VEL
LIN {X 0,Y 419.771,Z 372.698,A -85,B 0,C 180,E1 20604.23,E2 20604.23} C_VEL
LIN {X 0,Y 417.494,Z 372.979,A -85,B 0,C 180,E1 20602.884,E2 20602.884} C_VEL
LIN {X 0,Y 417.326,Z 373,A -85,B 0,C 180,E1 20602.5,E2 20602.5} C_VEL
LIN {X 0,Y 417.344,Z 373.002,A -85,B 0,C 180,E1 20598.671,E2 20598.671} C_VEL
LIN {X 0,Y 417.359,Z 372.996,A -85,B 0,C 180,E1 20594.721,E2 20594.721} C_VEL
LIN {X 0,Y 417.346,Z 372.999,A -85,B 0,C 180,E1 20590.84,E2 20590.84} C_VEL
LIN {X 0,Y 417.317,Z 373.004,A -85,B 0,C 180,E1 20587.162,E2 20587.162} C_VEL
LIN {X 0,Y 417.307,Z 373.003,A -85,B 0,C 180,E1 20583.382,E2 20583.382} C_VEL
LIN {X 0,Y 417.304,Z 373.002,A -85,B 0,C 180,E1 20579.586,E2 20579.586} C_VEL
LIN {X 0,Y 417.318,Z 373.003,A -85,B 0,C 180,E1 20575.901,E2 20575.901} C_VEL
LIN {X 0,Y 417.343,Z 373.002,A -85,B 0,C 180,E1 20572.172,E2 20572.172} C_VEL
LIN {X 0,Y 417.36,Z 372.998,A -85,B 0,C 180,E1 20568.356,E2 20568.356} C_VEL
LIN {X 0,Y 417.35,Z 372.998,A -85,B 0,C 180,E1 20564.379,E2 20564.379} C_VEL
LIN {X 0,Y 417.331,Z 372.999,A -85,B 0,C 180,E1 20560.583,E2 20560.583} C_VEL
LIN {X 0,Y 417.311,Z 373.001,A -85,B 0,C 180,E1 20556.848,E2 20556.848} C_VEL
LIN {X 0,Y 417.306,Z 373.003,A -85,B 0,C 180,E1 20553.011,E2 20553.011} C_VEL
LIN {X 0,Y 417.308,Z 373.002,A -85,B 0,C 180,E1 20549.094,E2 20549.094} C_VEL
LIN {X 0,Y 417.317,Z 372.979,A -85,B 0,C 180,E1 20545.387,E2 20545.387} C_VEL
LIN {X 0,Y 417.342,Z 372.992,A -85,B 0,C 180,E1 20541.638,E2 20541.638} C_VEL
LIN {X 0,Y 417.351,Z 372.958,A -85,B 0,C 180,E1 20537.85,E2 20537.85} C_VEL
LIN {X 0,Y 417.345,Z 372.995,A -85,B 0,C 180,E1 20533.996,E2 20533.996} C_VEL
LIN {X 0,Y 417.317,Z 372.96,A -85,B 0,C 180,E1 20530.206,E2 20530.206} C_VEL
LIN {X 0,Y 417.308,Z 372.997,A -85,B 0,C 180,E1 20526.459,E2 20526.459} C_VEL
LIN {X 0,Y 417.303,Z 372.965,A -85,B 0,C 180,E1 20522.603,E2 20522.603} C_VEL
LIN {X 0,Y 417.311,Z 372.998,A -85,B 0,C 180,E1 20518.759,E2 20518.759} C_VEL
LIN {X 0,Y 417.327,Z 372.971,A -85,B 0,C 180,E1 20515.046,E2 20515.046} C_VEL
LIN {X 0,Y 417.356,Z 372.981,A -85,B 0,C 180,E1 20511.314,E2 20511.314} C_VEL
LIN {X 0,Y 417.353,Z 372.969,A -85,B 0,C 180,E1 20507.403,E2 20507.403} C_VEL
LIN {X 0,Y 417.329,Z 372.986,A -85,B 0,C 180,E1 20503.716,E2 20503.716} C_VEL
LIN {X 0,Y 417.314,Z 372.974,A -85,B 0,C 180,E1 20499.914,E2 20499.914} C_VEL
LIN {X 0,Y 417.311,Z 372.999,A -85,B 0,C 180,E1 20496.109,E2 20496.109} C_VEL
LIN {X 0,Y 417.31,Z 372.964,A -85,B 0,C 180,E1 20492.297,E2 20492.297} C_VEL
LIN {X 0,Y 417.327,Z 372.998,A -85,B 0,C 180,E1 20488.529,E2 20488.529} C_VEL
LIN {X 0,Y 417.346,Z 372.998,A -85,B 0,C 180,E1 20484.729,E2 20484.729} C_VEL
LIN {X 0,Y 417.369,Z 372.989,A -85,B 0,C 180,E1 20480.91,E2 20480.91} C_VEL
LIN {X 0,Y 417.358,Z 372.997,A -85,B 0,C 180,E1 20476.942,E2 20476.942} C_VEL
LIN {X 0,Y 417.354,Z 373.286,A -85,B 0,C 180,E1 20475.749,E2 20475.749} C_VEL
LIN {X 0,Y 421.882,Z 387.317,A -85,B 0,C 180,E1 20472.413,E2 20472.413} C_VEL
LIN {X 0,Y 422.886,Z 390.227,A -85,B 0,C 180,E1 20471.839,E2 20471.839} C_VEL
LIN {X 0,Y 433.726,Z 409.466,A -85,B 0,C 180,E1 20470.16,E2 20470.16} C_VEL
LIN {X 0,Y 442.259,Z 425.844,A -85,B 0,C 180,E1 20468.906,E2 20468.906} C_VEL
LIN {X 0,Y 445.052,Z 437.8,A -85,B 0,C 180,E1 20468.378,E2 20468.378} C_VEL
LIN {X 0,Y 439.617,Z 648.488,A -85,B 0,C 180,E1 20464.693,E2 20464.693} C_VEL
LIN {X 0,Y 438.394,Z 669.367,A -85,B 0,C 180,E1 20464.143,E2 20464.143} C_VEL
LIN {X 0,Y 436.83,Z 688.001,A -85,B 0,C 180,E1 20463.424,E2 20463.424} C_VEL
LIN {X 0,Y 435.199,Z 704.396,A -85,B 0,C 180,E1 20462.618,E2 20462.618} C_VEL
LIN {X 0,Y 433.022,Z 723.557,A -85,B 0,C 180,E1 20461.455,E2 20461.455} C_VEL
LIN {X 0,Y 430.682,Z 741.321,A -85,B 0,C 180,E1 20460.096,E2 20460.096} C_VEL
LIN {X 0,Y 428.663,Z 755.762,A -85,B 0,C 180,E1 20458.793,E2 20458.793} C_VEL
LIN {X 0,Y 426.297,Z 772.161,A -85,B 0,C 180,E1 20457.065,E2 20457.065} C_VEL
LIN {X 0,Y 423.922,Z 787.78,A -85,B 0,C 180,E1 20455.077,E2 20455.077} C_VEL
LIN {X 0,Y 422.145,Z 799.814,A -85,B 0,C 180,E1 20453.299,E2 20453.299} C_VEL
LIN {X 0,Y 420.308,Z 812.969,A -85,B 0,C 180,E1 20451.051,E2 20451.051} C_VEL
LIN {X 0,Y 418.768,Z 824.56,A -85,B 0,C 180,E1 20448.659,E2 20448.659} C_VEL
LIN {X 0,Y 417.759,Z 833.31,A -85,B 0,C 180,E1 20446.547,E2 20446.547} C_VEL
LIN {X 0,Y 416.909,Z 842.191,A -85,B 0,C 180,E1 20444.017,E2 20444.017} C_VEL
LIN {X 0,Y 416.348,Z 849.592,A -85,B 0,C 180,E1 20441.357,E2 20441.357} C_VEL
LIN {X 0,Y 416.088,Z 854.814,A -85,B 0,C 180,E1 20438.986,E2 20438.986} C_VEL
LIN {X 0,Y 415.962,Z 858.787,A -85,B 0,C 180,E1 20436.625,E2 20436.625} C_VEL
LIN {X 0,Y 415.928,Z 862.017,A -85,B 0,C 180,E1 20433.721,E2 20433.721} C_VEL
LIN {X 0,Y 415.927,Z 863.278,A -85,B 0,C 180,E1 20431.24,E2 20431.24} C_VEL
LIN {X 0,Y 415.93,Z 863.337,A -85,B 0,C 180,E1 20429.036,E2 20429.036} C_VEL
LIN {X 0,Y 415.927,Z 862.284,A -85,B 0,C 180,E1 20426.693,E2 20426.693} C_VEL
LIN {X 0,Y 415.951,Z 859.616,A -85,B 0,C 180,E1 20423.929,E2 20423.929} C_VEL
LIN {X 0,Y 416.065,Z 855.356,A -85,B 0,C 180,E1 20421.292,E2 20421.292} C_VEL
LIN {X 0,Y 416.31,Z 850.263,A -85,B 0,C 180,E1 20418.923,E2 20418.923} C_VEL
LIN {X 0,Y 416.797,Z 843.462,A -85,B 0,C 180,E1 20416.403,E2 20416.403} C_VEL
LIN {X 0,Y 417.649,Z 834.397,A -85,B 0,C 180,E1 20413.734,E2 20413.734} C_VEL
LIN {X 0,Y 418.618,Z 825.803,A -85,B 0,C 180,E1 20411.623,E2 20411.623} C_VEL
LIN {X 0,Y 419.901,Z 815.805,A -85,B 0,C 180,E1 20409.511,E2 20409.511} C_VEL
LIN {X 0,Y 421.772,Z 802.494,A -85,B 0,C 180,E1 20407.122,E2 20407.122} C_VEL
LIN {X 0,Y 423.716,Z 789.125,A -85,B 0,C 180,E1 20405.11,E2 20405.11} C_VEL
LIN {X 0,Y 425.762,Z 775.585,A -85,B 0,C 180,E1 20403.351,E2 20403.351} C_VEL
LIN {X 0,Y 428.362,Z 757.9,A -85,B 0,C 180,E1 20401.413,E2 20401.413} C_VEL
LIN {X 0,Y 430.458,Z 742.937,A -85,B 0,C 180,E1 20400.041,E2 20400.041} C_VEL
LIN {X 0,Y 432.527,Z 727.26,A -85,B 0,C 180,E1 20398.815,E2 20398.815} C_VEL
LIN {X 0,Y 434.963,Z 706.69,A -85,B 0,C 180,E1 20397.506,E2 20397.506} C_VEL
LIN {X 0,Y 436.647,Z 689.961,A -85,B 0,C 180,E1 20396.664,E2 20396.664} C_VEL
LIN {X 0,Y 438.101,Z 673.031,A -85,B 0,C 180,E1 20395.989,E2 20395.989} C_VEL
LIN {X 0,Y 439.472,Z 652.084,A -85,B 0,C 180,E1 20395.38,E2 20395.38} C_VEL
LIN {X 0,Y 440.654,Z 611.487,A -85,B 0,C 180,E1 20394.639,E2 20394.639} C_VEL
LIN {X 0,Y 444.956,Z 436.627,A -85,B 0,C 180,E1 20391.589,E2 20391.589} C_VEL
LIN {X 0,Y 441.801,Z 424.831,A -85,B 0,C 180,E1 20391.026,E2 20391.026} C_VEL
LIN {X 0,Y 431.146,Z 404.68,A -85,B 0,C 180,E1 20389.449,E2 20389.449} C_VEL
LIN {X 0,Y 422.634,Z 389.58,A -85,B 0,C 180,E1 20388.081,E2 20388.081} C_VEL
LIN {X 0,Y 418.175,Z 375.701,A -85,B 0,C 180,E1 20384.862,E2 20384.862} C_VEL
LIN {X 0,Y 417.324,Z 373.081,A -85,B 0,C 180,E1 20384.157,E2 20384.157} C_VEL
LIN {X 0,Y 417.313,Z 372.998,A -85,B 0,C 180,E1 20380.313,E2 20380.313} C_VEL
LIN {X 0,Y 417.331,Z 372.99,A -85,B 0,C 180,E1 20376.623,E2 20376.623} C_VEL
LIN {X 0,Y 417.358,Z 372.975,A -85,B 0,C 180,E1 20372.949,E2 20372.949} C_VEL
LIN {X 0,Y 417.353,Z 372.97,A -85,B 0,C 180,E1 20369.104,E2 20369.104} C_VEL
LIN {X 0,Y 417.335,Z 372.997,A -85,B 0,C 180,E1 20365.247,E2 20365.247} C_VEL
LIN {X 0,Y 417.311,Z 372.962,A -85,B 0,C 180,E1 20361.51,E2 20361.51} C_VEL
LIN {X 0,Y 417.308,Z 373.002,A -85,B 0,C 180,E1 20357.72,E2 20357.72} C_VEL
LIN {X 0,Y 417.305,Z 372.959,A -85,B 0,C 180,E1 20353.868,E2 20353.868} C_VEL
LIN {X 0,Y 417.323,Z 373,A -85,B 0,C 180,E1 20350.078,E2 20350.078} C_VEL
LIN {X 0,Y 417.34,Z 372.953,A -85,B 0,C 180,E1 20346.333,E2 20346.333} C_VEL
LIN {X 0,Y 417.355,Z 373,A -85,B 0,C 180,E1 20342.477,E2 20342.477} C_VEL
LIN {X 0,Y 417.34,Z 372.952,A -85,B 0,C 180,E1 20338.633,E2 20338.633} C_VEL
LIN {X 0,Y 417.33,Z 372.998,A -85,B 0,C 180,E1 20334.783,E2 20334.783} C_VEL
LIN {X 0,Y 417.307,Z 372.959,A -85,B 0,C 180,E1 20331.047,E2 20331.047} C_VEL
LIN {X 0,Y 417.306,Z 373.001,A -85,B 0,C 180,E1 20327.197,E2 20327.197} C_VEL
LIN {X 0,Y 417.302,Z 372.959,A -85,B 0,C 180,E1 20323.298,E2 20323.298} C_VEL
LIN {X 0,Y 417.316,Z 373.002,A -85,B 0,C 180,E1 20319.517,E2 20319.517} C_VEL
LIN {X 0,Y 417.337,Z 372.962,A -85,B 0,C 180,E1 20315.824,E2 20315.824} C_VEL
LIN {X 0,Y 417.359,Z 372.999,A -85,B 0,C 180,E1 20312.004,E2 20312.004} C_VEL
LIN {X 0,Y 417.341,Z 373.001,A -85,B 0,C 180,E1 20308.202,E2 20308.202} C_VEL
LIN {X 0,Y 417.32,Z 373.003,A -85,B 0,C 180,E1 20304.405,E2 20304.405} C_VEL
LIN {X 0,Y 417.305,Z 373.001,A -85,B 0,C 180,E1 20300.704,E2 20300.704} C_VEL
LIN {X 0,Y 417.308,Z 373.004,A -85,B 0,C 180,E1 20296.945,E2 20296.945} C_VEL
LIN {X 0,Y 417.325,Z 373.004,A -85,B 0,C 180,E1 20293.251,E2 20293.251} C_VEL
LIN {X 0,Y 417.355,Z 373,A -85,B 0,C 180,E1 20289.533,E2 20289.533} C_VEL
LIN {X 0,Y 417.352,Z 372.997,A -85,B 0,C 180,E1 20285.601,E2 20285.601} C_VEL
LIN {X 0,Y 417.342,Z 372.998,A -85,B 0,C 180,E1 20281.752,E2 20281.752} C_VEL
LIN {X 0,Y 417.317,Z 373.003,A -85,B 0,C 180,E1 20278.007,E2 20278.007} C_VEL
LIN {X 0,Y 417.308,Z 373.005,A -85,B 0,C 180,E1 20274.186,E2 20274.186} C_VEL
LIN {X 0,Y 417.302,Z 373.002,A -85,B 0,C 180,E1 20270.329,E2 20270.329} C_VEL
LIN {X 0,Y 417.305,Z 373.006,A -85,B 0,C 180,E1 20266.423,E2 20266.423} C_VEL
LIN {X 0,Y 417.32,Z 373.002,A -85,B 0,C 180,E1 20262.734,E2 20262.734} C_VEL
LIN {X 0,Y 417.342,Z 372.998,A -85,B 0,C 180,E1 20258.959,E2 20258.959} C_VEL
LIN {X 0,Y 417.345,Z 372.999,A -85,B 0,C 180,E1 20255.223,E2 20255.223} C_VEL
LIN {X 0,Y 417.328,Z 373.002,A -85,B 0,C 180,E1 20251.373,E2 20251.373} C_VEL
LIN {X 0,Y 417.306,Z 373.002,A -85,B 0,C 180,E1 20247.666,E2 20247.666} C_VEL
LIN {X 0,Y 417.303,Z 373.005,A -85,B 0,C 180,E1 20243.807,E2 20243.807} C_VEL
LIN {X 0,Y 417.326,Z 373,A -85,B 0,C 180,E1 20242.5,E2 20242.5} C_VEL
LIN {X 0,Y 416.286,Z 373.133,A -85,B 0,C 180,E1 20241.443,E2 20241.443} C_VEL
LIN {X 0,Y 409.793,Z 373.94,A -85,B 0,C 180,E1 20238.386,E2 20238.386} C_VEL
LIN {X 0,Y 409.365,Z 373.991,A -85,B 0,C 180,E1 20237.685,E2 20237.685} C_VEL
LIN {X 0,Y 409.365,Z 373.995,A -85,B 0,C 180,E1 20233.833,E2 20233.833} C_VEL
LIN {X 0,Y 409.371,Z 373.991,A -85,B 0,C 180,E1 20230.006,E2 20230.006} C_VEL
LIN {X 0,Y 409.391,Z 373.988,A -85,B 0,C 180,E1 20226.236,E2 20226.236} C_VEL
LIN {X 0,Y 409.407,Z 373.99,A -85,B 0,C 180,E1 20222.354,E2 20222.354} C_VEL
LIN {X 0,Y 409.416,Z 373.986,A -85,B 0,C 180,E1 20218.446,E2 20218.446} C_VEL
LIN {X 0,Y 409.413,Z 373.986,A -85,B 0,C 180,E1 20214.464,E2 20214.464} C_VEL
LIN {X 0,Y 409.413,Z 373.989,A -85,B 0,C 180,E1 20210.495,E2 20210.495} C_VEL
LIN {X 0,Y 409.392,Z 373.991,A -85,B 0,C 180,E1 20206.665,E2 20206.665} C_VEL
LIN {X 0,Y 409.375,Z 373.991,A -85,B 0,C 180,E1 20202.887,E2 20202.887} C_VEL
LIN {X 0,Y 409.367,Z 373.99,A -85,B 0,C 180,E1 20199.043,E2 20199.043} C_VEL
LIN {X 0,Y 409.368,Z 373.993,A -85,B 0,C 180,E1 20195.096,E2 20195.096} C_VEL
LIN {X 0,Y 409.369,Z 373.991,A -85,B 0,C 180,E1 20191.175,E2 20191.175} C_VEL
LIN {X 0,Y 409.384,Z 373.992,A -85,B 0,C 180,E1 20187.482,E2 20187.482} C_VEL
LIN {X 0,Y 409.393,Z 373.951,A -85,B 0,C 180,E1 20183.603,E2 20183.603} C_VEL
LIN {X 0,Y 409.416,Z 373.981,A -85,B 0,C 180,E1 20179.836,E2 20179.836} C_VEL
LIN {X 0,Y 409.417,Z 373.951,A -85,B 0,C 180,E1 20175.808,E2 20175.808} C_VEL
LIN {X 0,Y 409.403,Z 373.976,A -85,B 0,C 180,E1 20171.974,E2 20171.974} C_VEL
LIN {X 0,Y 409.383,Z 373.955,A -85,B 0,C 180,E1 20168.137,E2 20168.137} C_VEL
LIN {X 0,Y 409.374,Z 373.984,A -85,B 0,C 180,E1 20164.336,E2 20164.336} C_VEL
LIN {X 0,Y 409.365,Z 373.951,A -85,B 0,C 180,E1 20160.554,E2 20160.554} C_VEL
LIN {X 0,Y 409.369,Z 373.987,A -85,B 0,C 180,E1 20156.634,E2 20156.634} C_VEL
LIN {X 0,Y 409.375,Z 373.947,A -85,B 0,C 180,E1 20152.839,E2 20152.839} C_VEL
LIN {X 0,Y 409.399,Z 373.985,A -85,B 0,C 180,E1 20149.039,E2 20149.039} C_VEL
LIN {X 0,Y 409.411,Z 373.944,A -85,B 0,C 180,E1 20145.136,E2 20145.136} C_VEL
LIN {X 0,Y 409.417,Z 373.978,A -85,B 0,C 180,E1 20141.189,E2 20141.189} C_VEL
LIN {X 0,Y 409.415,Z 373.958,A -85,B 0,C 180,E1 20137.298,E2 20137.298} C_VEL
LIN {X 0,Y 409.396,Z 373.962,A -85,B 0,C 180,E1 20133.448,E2 20133.448} C_VEL
LIN {X 0,Y 409.384,Z 373.988,A -85,B 0,C 180,E1 20129.626,E2 20129.626} C_VEL
LIN {X 0,Y 409.372,Z 373.973,A -85,B 0,C 180,E1 20125.818,E2 20125.818} C_VEL
LIN {X 0,Y 409.371,Z 373.971,A -85,B 0,C 180,E1 20122.008,E2 20122.008} C_VEL
LIN {X 0,Y 409.378,Z 373.973,A -85,B 0,C 180,E1 20118.151,E2 20118.151} C_VEL
LIN {X 0,Y 409.448,Z 374.247,A -85,B 0,C 180,E1 20116.618,E2 20116.618} C_VEL
LIN {X 0,Y 413.8,Z 387.53,A -85,B 0,C 180,E1 20113.33,E2 20113.33} C_VEL
LIN {X 0,Y 414.604,Z 389.884,A -85,B 0,C 180,E1 20112.872,E2 20112.872} C_VEL
LIN {X 0,Y 426.835,Z 411.057,A -85,B 0,C 180,E1 20110.905,E2 20110.905} C_VEL
LIN {X 0,Y 436.548,Z 429.938,A -85,B 0,C 180,E1 20109.424,E2 20109.424} C_VEL
LIN {X 0,Y 438.726,Z 439.714,A -85,B 0,C 180,E1 20108.991,E2 20108.991} C_VEL
LIN {X 0,Y 433.041,Z 648.251,A -85,B 0,C 180,E1 20105.298,E2 20105.298} C_VEL
LIN {X 0,Y 431.76,Z 669.143,A -85,B 0,C 180,E1 20104.741,E2 20104.741} C_VEL
LIN {X 0,Y 430.075,Z 688.229,A -85,B 0,C 180,E1 20103.994,E2 20103.994} C_VEL
LIN {X 0,Y 428.339,Z 704.815,A -85,B 0,C 180,E1 20103.165,E2 20103.165} C_VEL
LIN {X 0,Y 425.987,Z 724.253,A -85,B 0,C 180,E1 20101.956,E2 20101.956} C_VEL
LIN {X 0,Y 423.655,Z 741.081,A -85,B 0,C 180,E1 20100.648,E2 20100.648} C_VEL
LIN {X 0,Y 421.552,Z 755.342,A -85,B 0,C 180,E1 20099.345,E2 20099.345} C_VEL
LIN {X 0,Y 419.105,Z 771.287,A -85,B 0,C 180,E1 20097.646,E2 20097.646} C_VEL
LIN {X 0,Y 416.552,Z 787.244,A -85,B 0,C 180,E1 20095.597,E2 20095.597} C_VEL
LIN {X 0,Y 414.606,Z 799.571,A -85,B 0,C 180,E1 20093.748,E2 20093.748} C_VEL
LIN {X 0,Y 412.645,Z 812.726,A -85,B 0,C 180,E1 20091.461,E2 20091.461} C_VEL
LIN {X 0,Y 410.996,Z 824.318,A -85,B 0,C 180,E1 20089.025,E2 20089.025} C_VEL
LIN {X 0,Y 409.911,Z 833.068,A -85,B 0,C 180,E1 20086.873,E2 20086.873} C_VEL
LIN {X 0,Y 408.996,Z 841.95,A -85,B 0,C 180,E1 20084.294,E2 20084.294} C_VEL
LIN {X 0,Y 408.384,Z 849.352,A -85,B 0,C 180,E1 20081.581,E2 20081.581} C_VEL
LIN {X 0,Y 408.102,Z 854.575,A -85,B 0,C 180,E1 20079.163,E2 20079.163} C_VEL
LIN {X 0,Y 407.969,Z 858.55,A -85,B 0,C 180,E1 20076.756,E2 20076.756} C_VEL
LIN {X 0,Y 407.929,Z 861.78,A -85,B 0,C 180,E1 20073.794,E2 20073.794} C_VEL
LIN {X 0,Y 407.93,Z 863.042,A -85,B 0,C 180,E1 20071.264,E2 20071.264} C_VEL
LIN {X 0,Y 407.933,Z 863.101,A -85,B 0,C 180,E1 20069.017,E2 20069.017} C_VEL
LIN {X 0,Y 407.929,Z 862.047,A -85,B 0,C 180,E1 20066.628,E2 20066.628} C_VEL
LIN {X 0,Y 407.952,Z 859.378,A -85,B 0,C 180,E1 20063.809,E2 20063.809} C_VEL
LIN {X 0,Y 408.079,Z 855.117,A -85,B 0,C 180,E1 20061.121,E2 20061.121} C_VEL
LIN {X 0,Y 408.341,Z 850.023,A -85,B 0,C 180,E1 20058.704,E2 20058.704} C_VEL
LIN {X 0,Y 408.87,Z 843.221,A -85,B 0,C 180,E1 20056.134,E2 20056.134} C_VEL
LIN {X 0,Y 409.791,Z 834.155,A -85,B 0,C 180,E1 20053.414,E2 20053.414} C_VEL
LIN {X 0,Y 410.864,Z 825.322,A -85,B 0,C 180,E1 20051.207,E2 20051.207} C_VEL
LIN {X 0,Y 412.276,Z 815.144,A -85,B 0,C 180,E1 20049.026,E2 20049.026} C_VEL
LIN {X 0,Y 414.397,Z 800.986,A -85,B 0,C 180,E1 20046.478,E2 20046.478} C_VEL
LIN {X 0,Y 416.388,Z 788.243,A -85,B 0,C 180,E1 20044.544,E2 20044.544} C_VEL
LIN {X 0,Y 418.683,Z 773.962,A -85,B 0,C 180,E1 20042.674,E2 20042.674} C_VEL
LIN {X 0,Y 421.313,Z 756.947,A -85,B 0,C 180,E1 20040.812,E2 20040.812} C_VEL
LIN {X 0,Y 423.421,Z 742.696,A -85,B 0,C 180,E1 20039.49,E2 20039.49} C_VEL
LIN {X 0,Y 425.596,Z 727.02,A -85,B 0,C 180,E1 20038.249,E2 20038.249} C_VEL
LIN {X 0,Y 428.167,Z 706.409,A -85,B 0,C 180,E1 20036.922,E2 20036.922} C_VEL
LIN {X 0,Y 429.931,Z 689.723,A -85,B 0,C 180,E1 20036.073,E2 20036.073} C_VEL
LIN {X 0,Y 431.463,Z 672.659,A -85,B 0,C 180,E1 20035.386,E2 20035.386} C_VEL
LIN {X 0,Y 432.908,Z 651.436,A -85,B 0,C 180,E1 20034.768,E2 20034.768} C_VEL
LIN {X 0,Y 434.192,Z 608.955,A -85,B 0,C 180,E1 20033.986,E2 20033.986} C_VEL
LIN {X 0,Y 438.651,Z 438.5,A -85,B 0,C 180,E1 20030.977,E2 20030.977} C_VEL
LIN {X 0,Y 436.054,Z 428.834,A -85,B 0,C 180,E1 20030.5,E2 20030.5} C_VEL
LIN {X 0,Y 425.835,Z 409.362,A -85,B 0,C 180,E1 20028.942,E2 20028.942} C_VEL
LIN {X 0,Y 416.657,Z 393.562,A -85,B 0,C 180,E1 20027.482,E2 20027.482} C_VEL
LIN {X 0,Y 414.321,Z 389.232,A -85,B 0,C 180,E1 20027.043,E2 20027.043} C_VEL
LIN {X 0,Y 410.199,Z 376.67,A -85,B 0,C 180,E1 20024.007,E2 20024.007} C_VEL
LIN {X 0,Y 409.426,Z 374.058,A -85,B 0,C 180,E1 20023.304,E2 20023.304} C_VEL
LIN {X 0,Y 409.402,Z 373.987,A -85,B 0,C 180,E1 20019.423,E2 20019.423} C_VEL
LIN {X 0,Y 409.388,Z 373.992,A -85,B 0,C 180,E1 20015.545,E2 20015.545} C_VEL
LIN {X 0,Y 409.375,Z 373.986,A -85,B 0,C 180,E1 20011.796,E2 20011.796} C_VEL
LIN {X 0,Y 409.369,Z 373.952,A -85,B 0,C 180,E1 20007.971,E2 20007.971} C_VEL
LIN {X 0,Y 409.374,Z 373.988,A -85,B 0,C 180,E1 20004.077,E2 20004.077} C_VEL
LIN {X 0,Y 409.384,Z 373.956,A -85,B 0,C 180,E1 20000.297,E2 20000.297} C_VEL
LIN {X 0,Y 409.402,Z 373.975,A -85,B 0,C 180,E1 19996.462,E2 19996.462} C_VEL
LIN {X 0,Y 409.414,Z 373.955,A -85,B 0,C 180,E1 19992.702,E2 19992.702} C_VEL
LIN {X 0,Y 409.415,Z 373.969,A -85,B 0,C 180,E1 19988.714,E2 19988.714} C_VEL
LIN {X 0,Y 409.395,Z 373.959,A -85,B 0,C 180,E1 19984.849,E2 19984.849} C_VEL
LIN {X 0,Y 409.377,Z 373.982,A -85,B 0,C 180,E1 19981.126,E2 19981.126} C_VEL
LIN {X 0,Y 409.365,Z 373.952,A -85,B 0,C 180,E1 19977.346,E2 19977.346} C_VEL
LIN {X 0,Y 409.367,Z 373.986,A -85,B 0,C 180,E1 19973.415,E2 19973.415} C_VEL
LIN {X 0,Y 409.369,Z 373.951,A -85,B 0,C 180,E1 19969.594,E2 19969.594} C_VEL
LIN {X 0,Y 409.39,Z 373.984,A -85,B 0,C 180,E1 19965.829,E2 19965.829} C_VEL
LIN {X 0,Y 409.41,Z 373.946,A -85,B 0,C 180,E1 19962.086,E2 19962.086} C_VEL
LIN {X 0,Y 409.423,Z 373.973,A -85,B 0,C 180,E1 19958.121,E2 19958.121} C_VEL
LIN {X 0,Y 409.405,Z 373.97,A -85,B 0,C 180,E1 19954.242,E2 19954.242} C_VEL
LIN {X 0,Y 409.391,Z 373.991,A -85,B 0,C 180,E1 19950.393,E2 19950.393} C_VEL
LIN {X 0,Y 409.373,Z 373.992,A -85,B 0,C 180,E1 19946.645,E2 19946.645} C_VEL
LIN {X 0,Y 409.368,Z 373.989,A -85,B 0,C 180,E1 19942.73,E2 19942.73} C_VEL
LIN {X 0,Y 409.365,Z 373.992,A -85,B 0,C 180,E1 19938.786,E2 19938.786} C_VEL
LIN {X 0,Y 409.369,Z 373.993,A -85,B 0,C 180,E1 19934.898,E2 19934.898} C_VEL
LIN {X 0,Y 409.377,Z 373.991,A -85,B 0,C 180,E1 19931.015,E2 19931.015} C_VEL
LIN {X 0,Y 409.391,Z 373.988,A -85,B 0,C 180,E1 19927.248,E2 19927.248} C_VEL
LIN {X 0,Y 409.409,Z 373.987,A -85,B 0,C 180,E1 19923.377,E2 19923.377} C_VEL
LIN {X 0,Y 409.42,Z 373.988,A -85,B 0,C 180,E1 19919.557,E2 19919.557} C_VEL
LIN {X 0,Y 409.403,Z 373.988,A -85,B 0,C 180,E1 19915.611,E2 19915.611} C_VEL
LIN {X 0,Y 409.385,Z 373.989,A -85,B 0,C 180,E1 19911.791,E2 19911.791} C_VEL
LIN {X 0,Y 409.368,Z 373.994,A -85,B 0,C 180,E1 19908.07,E2 19908.07} C_VEL
LIN {X 0,Y 409.363,Z 373.993,A -85,B 0,C 180,E1 19904.191,E2 19904.191} C_VEL
LIN {X 0,Y 409.364,Z 373.992,A -85,B 0,C 180,E1 19900.219,E2 19900.219} C_VEL
LIN {X 0,Y 409.366,Z 373.994,A -85,B 0,C 180,E1 19896.31,E2 19896.31} C_VEL
LIN {X 0,Y 409.377,Z 373.99,A -85,B 0,C 180,E1 19892.52,E2 19892.52} C_VEL
LIN {X 0,Y 409.399,Z 373.989,A -85,B 0,C 180,E1 19888.741,E2 19888.741} C_VEL
LIN {X 0,Y 409.408,Z 373.988,A -85,B 0,C 180,E1 19884.816,E2 19884.816} C_VEL
LIN {X 0,Y 409.405,Z 373.986,A -85,B 0,C 180,E1 19881.008,E2 19881.008} C_VEL
LIN {X 0,Y 409.365,Z 373.991,A -85,B 0,C 180,E1 19877.685,E2 19877.685} C_VEL
LIN {X 0,Y 408.376,Z 374.117,A -85,B 0,C 180,E1 19876.606,E2 19876.606} C_VEL
LIN {X 0,Y 401.872,Z 374.927,A -85,B 0,C 180,E1 19873.487,E2 19873.487} C_VEL
LIN {X 0,Y 401.471,Z 374.975,A -85,B 0,C 180,E1 19872.772,E2 19872.772} C_VEL
LIN {X 0,Y 401.468,Z 374.98,A -85,B 0,C 180,E1 19868.831,E2 19868.831} C_VEL
LIN {X 0,Y 401.453,Z 374.977,A -85,B 0,C 180,E1 19864.951,E2 19864.951} C_VEL
LIN {X 0,Y 401.438,Z 374.979,A -85,B 0,C 180,E1 19861.107,E2 19861.107} C_VEL
LIN {X 0,Y 401.43,Z 374.983,A -85,B 0,C 180,E1 19857.284,E2 19857.284} C_VEL
LIN {X 0,Y 401.429,Z 374.981,A -85,B 0,C 180,E1 19853.308,E2 19853.308} C_VEL
LIN {X 0,Y 401.427,Z 374.979,A -85,B 0,C 180,E1 19849.422,E2 19849.422} C_VEL
LIN {X 0,Y 401.434,Z 374.981,A -85,B 0,C 180,E1 19845.583,E2 19845.583} C_VEL
LIN {X 0,Y 401.452,Z 374.981,A -85,B 0,C 180,E1 19841.861,E2 19841.861} C_VEL
LIN {X 0,Y 401.478,Z 374.978,A -85,B 0,C 180,E1 19838.098,E2 19838.098} C_VEL
LIN {X 0,Y 401.474,Z 374.979,A -85,B 0,C 180,E1 19834.07,E2 19834.07} C_VEL
LIN {X 0,Y 401.489,Z 374.976,A -85,B 0,C 180,E1 19830.028,E2 19830.028} C_VEL
LIN {X 0,Y 401.474,Z 374.961,A -85,B 0,C 180,E1 19825.969,E2 19825.969} C_VEL
LIN {X 0,Y 401.487,Z 374.96,A -85,B 0,C 180,E1 19821.927,E2 19821.927} C_VEL
LIN {X 0,Y 401.468,Z 374.934,A -85,B 0,C 180,E1 19817.947,E2 19817.947} C_VEL
LIN {X 0,Y 401.469,Z 374.973,A -85,B 0,C 180,E1 19813.972,E2 19813.972} C_VEL
LIN {X 0,Y 401.451,Z 374.931,A -85,B 0,C 180,E1 19810.033,E2 19810.033} C_VEL
LIN {X 0,Y 401.437,Z 374.975,A -85,B 0,C 180,E1 19806.285,E2 19806.285} C_VEL
LIN {X 0,Y 401.426,Z 374.935,A -85,B 0,C 180,E1 19802.42,E2 19802.42} C_VEL
LIN {X 0,Y 401.431,Z 374.976,A -85,B 0,C 180,E1 19798.567,E2 19798.567} C_VEL
LIN {X 0,Y 401.43,Z 374.94,A -85,B 0,C 180,E1 19794.706,E2 19794.706} C_VEL
LIN {X 0,Y 401.451,Z 374.967,A -85,B 0,C 180,E1 19790.967,E2 19790.967} C_VEL
LIN {X 0,Y 401.469,Z 374.941,A -85,B 0,C 180,E1 19787.188,E2 19787.188} C_VEL
LIN {X 0,Y 401.476,Z 374.964,A -85,B 0,C 180,E1 19783.352,E2 19783.352} C_VEL
LIN {X 0,Y 401.465,Z 374.937,A -85,B 0,C 180,E1 19779.436,E2 19779.436} C_VEL
LIN {X 0,Y 401.453,Z 374.978,A -85,B 0,C 180,E1 19775.574,E2 19775.574} C_VEL
LIN {X 0,Y 401.438,Z 374.94,A -85,B 0,C 180,E1 19771.751,E2 19771.751} C_VEL
LIN {X 0,Y 401.433,Z 374.968,A -85,B 0,C 180,E1 19767.954,E2 19767.954} C_VEL
LIN {X 0,Y 401.435,Z 374.981,A -85,B 0,C 180,E1 19763.994,E2 19763.994} C_VEL
LIN {X 0,Y 401.435,Z 374.981,A -85,B 0,C 180,E1 19760.009,E2 19760.009} C_VEL
LIN {X 0,Y 401.471,Z 375.198,A -85,B 0,C 180,E1 19757.547,E2 19757.547} C_VEL
LIN {X 0,Y 405.533,Z 387.591,A -85,B 0,C 180,E1 19754.352,E2 19754.352} C_VEL
LIN {X 0,Y 406.336,Z 389.585,A -85,B 0,C 180,E1 19753.962,E2 19753.962} C_VEL
LIN {X 0,Y 416.808,Z 407.39,A -85,B 0,C 180,E1 19752.185,E2 19752.185} C_VEL
LIN {X 0,Y 427.049,Z 426.173,A -85,B 0,C 180,E1 19750.553,E2 19750.553} C_VEL
LIN {X 0,Y 431.018,Z 434.639,A -85,B 0,C 180,E1 19749.926,E2 19749.926} C_VEL
LIN {X 0,Y 432.455,Z 441.552,A -85,B 0,C 180,E1 19749.623,E2 19749.623} C_VEL
LIN {X 0,Y 426.517,Z 648.014,A -85,B 0,C 180,E1 19745.921,E2 19745.921} C_VEL
LIN {X 0,Y 425.173,Z 668.954,A -85,B 0,C 180,E1 19745.357,E2 19745.357} C_VEL
LIN {X 0,Y 423.464,Z 687.482,A -85,B 0,C 180,E1 19744.628,E2 19744.628} C_VEL
LIN {X 0,Y 421.773,Z 702.993,A -85,B 0,C 180,E1 19743.854,E2 19743.854} C_VEL
LIN {X 0,Y 419.671,Z 719.921,A -85,B 0,C 180,E1 19742.82,E2 19742.82} C_VEL
LIN {X 0,Y 416.919,Z 739.224,A -85,B 0,C 180,E1 19741.359,E2 19741.359} C_VEL
LIN {X 0,Y 414.532,Z 754.566,A -85,B 0,C 180,E1 19739.952,E2 19739.952} C_VEL
LIN {X 0,Y 412.069,Z 769.781,A -85,B 0,C 180,E1 19738.317,E2 19738.317} C_VEL
LIN {X 0,Y 409.342,Z 785.999,A -85,B 0,C 180,E1 19736.238,E2 19736.238} C_VEL
LIN {X 0,Y 407.241,Z 798.435,A -85,B 0,C 180,E1 19734.36,E2 19734.36} C_VEL
LIN {X 0,Y 405.357,Z 810.108,A -85,B 0,C 180,E1 19732.324,E2 19732.324} C_VEL
LIN {X 0,Y 403.377,Z 823.171,A -85,B 0,C 180,E1 19729.618,E2 19729.618} C_VEL
LIN {X 0,Y 402.107,Z 832.58,A -85,B 0,C 180,E1 19727.278,E2 19727.278} C_VEL
LIN {X 0,Y 401.134,Z 841.238,A -85,B 0,C 180,E1 19724.728,E2 19724.728} C_VEL
LIN {X 0,Y 400.424,Z 849.142,A -85,B 0,C 180,E1 19721.802,E2 19721.802} C_VEL
LIN {X 0,Y 400.118,Z 854.336,A -85,B 0,C 180,E1 19719.348,E2 19719.348} C_VEL
LIN {X 0,Y 399.977,Z 858.312,A -85,B 0,C 180,E1 19716.891,E2 19716.891} C_VEL
LIN {X 0,Y 399.931,Z 861.544,A -85,B 0,C 180,E1 19713.87,E2 19713.87} C_VEL
LIN {X 0,Y 399.932,Z 862.805,A -85,B 0,C 180,E1 19711.289,E2 19711.289} C_VEL
LIN {X 0,Y 399.936,Z 862.865,A -85,B 0,C 180,E1 19708.997,E2 19708.997} C_VEL
LIN {X 0,Y 399.931,Z 861.811,A -85,B 0,C 180,E1 19706.56,E2 19706.56} C_VEL
LIN {X 0,Y 399.954,Z 859.141,A -85,B 0,C 180,E1 19703.685,E2 19703.685} C_VEL
LIN {X 0,Y 400.095,Z 854.878,A -85,B 0,C 180,E1 19700.942,E2 19700.942} C_VEL
LIN {X 0,Y 400.376,Z 849.783,A -85,B 0,C 180,E1 19698.476,E2 19698.476} C_VEL
LIN {X 0,Y 400.954,Z 842.979,A -85,B 0,C 180,E1 19695.855,E2 19695.855} C_VEL
LIN {X 0,Y 401.944,Z 833.913,A -85,B 0,C 180,E1 19693.08,E2 19693.08} C_VEL
LIN {X 0,Y 403.066,Z 825.317,A -85,B 0,C 180,E1 19690.887,E2 19690.887} C_VEL
LIN {X 0,Y 404.542,Z 815.319,A -85,B 0,C 180,E1 19688.696,E2 19688.696} C_VEL
LIN {X 0,Y 406.766,Z 801.423,A -85,B 0,C 180,E1 19686.126,E2 19686.126} C_VEL
LIN {X 0,Y 408.874,Z 788.705,A -85,B 0,C 180,E1 19684.151,E2 19684.151} C_VEL
LIN {X 0,Y 411.08,Z 775.663,A -85,B 0,C 180,E1 19682.398,E2 19682.398} C_VEL
LIN {X 0,Y 413.875,Z 758.843,A -85,B 0,C 180,E1 19680.474,E2 19680.474} C_VEL
LIN {X 0,Y 416.303,Z 743.264,A -85,B 0,C 180,E1 19678.992,E2 19678.992} C_VEL
LIN {X 0,Y 418.554,Z 727.87,A -85,B 0,C 180,E1 19677.746,E2 19677.746} C_VEL
LIN {X 0,Y 421.089,Z 709.096,A -85,B 0,C 180,E1 19676.484,E2 19676.484} C_VEL
LIN {X 0,Y 423.188,Z 690.229,A -85,B 0,C 180,E1 19675.498,E2 19675.498} C_VEL
LIN {X 0,Y 424.774,Z 673.472,A -85,B 0,C 180,E1 19674.809,E2 19674.809} C_VEL
LIN {X 0,Y 426.285,Z 653.266,A -85,B 0,C 180,E1 19674.191,E2 19674.191} C_VEL
LIN {X 0,Y 427.478,Z 617.894,A -85,B 0,C 180,E1 19673.516,E2 19673.516} C_VEL
LIN {X 0,Y 432.363,Z 440.21,A -85,B 0,C 180,E1 19670.339,E2 19670.339} C_VEL
LIN {X 0,Y 430.346,Z 432.814,A -85,B 0,C 180,E1 19669.96,E2 19669.96} C_VEL
LIN {X 0,Y 419.183,Z 411.411,A -85,B 0,C 180,E1 19668.197,E2 19668.197} C_VEL
LIN {X 0,Y 408.601,Z 393.445,A -85,B 0,C 180,E1 19666.442,E2 19666.442} C_VEL
LIN {X 0,Y 405.99,Z 388.835,A -85,B 0,C 180,E1 19665.936,E2 19665.936} C_VEL
LIN {X 0,Y 402.156,Z 377.348,A -85,B 0,C 180,E1 19663.035,E2 19663.035} C_VEL
LIN {X 0,Y 401.444,Z 375.022,A -85,B 0,C 180,E1 19662.36,E2 19662.36} C_VEL
LIN {X 0,Y 401.444,Z 374.961,A -85,B 0,C 180,E1 19658.516,E2 19658.516} C_VEL
LIN {X 0,Y 401.462,Z 374.966,A -85,B 0,C 180,E1 19654.729,E2 19654.729} C_VEL
LIN {X 0,Y 401.475,Z 374.977,A -85,B 0,C 180,E1 19650.775,E2 19650.775} C_VEL
LIN {X 0,Y 401.473,Z 374.943,A -85,B 0,C 180,E1 19646.798,E2 19646.798} C_VEL
LIN {X 0,Y 401.484,Z 374.948,A -85,B 0,C 180,E1 19642.865,E2 19642.865} C_VEL
LIN {X 0,Y 401.476,Z 374.966,A -85,B 0,C 180,E1 19638.854,E2 19638.854} C_VEL
LIN {X 0,Y 401.472,Z 374.931,A -85,B 0,C 180,E1 19634.869,E2 19634.869} C_VEL
LIN {X 0,Y 401.463,Z 374.973,A -85,B 0,C 180,E1 19630.916,E2 19630.916} C_VEL
LIN {X 0,Y 401.436,Z 374.934,A -85,B 0,C 180,E1 19627.16,E2 19627.16} C_VEL
LIN {X 0,Y 401.432,Z 374.976,A -85,B 0,C 180,E1 19623.29,E2 19623.29} C_VEL
LIN {X 0,Y 401.426,Z 374.937,A -85,B 0,C 180,E1 19619.435,E2 19619.435} C_VEL
LIN {X 0,Y 401.431,Z 374.976,A -85,B 0,C 180,E1 19615.435,E2 19615.435} C_VEL
LIN {X 0,Y 401.429,Z 374.938,A -85,B 0,C 180,E1 19611.556,E2 19611.556} C_VEL
LIN {X 0,Y 401.447,Z 374.971,A -85,B 0,C 180,E1 19607.785,E2 19607.785} C_VEL
LIN {X 0,Y 401.46,Z 374.936,A -85,B 0,C 180,E1 19603.959,E2 19603.959} C_VEL
LIN {X 0,Y 401.476,Z 374.971,A -85,B 0,C 180,E1 19600.059,E2 19600.059} C_VEL
LIN {X 0,Y 401.468,Z 374.935,A -85,B 0,C 180,E1 19596.214,E2 19596.214} C_VEL
LIN {X 0,Y 401.465,Z 374.979,A -85,B 0,C 180,E1 19592.252,E2 19592.252} C_VEL
LIN {X 0,Y 401.444,Z 374.98,A -85,B 0,C 180,E1 19588.474,E2 19588.474} C_VEL
LIN {X 0,Y 401.431,Z 374.982,A -85,B 0,C 180,E1 19584.711,E2 19584.711} C_VEL
LIN {X 0,Y 401.427,Z 374.979,A -85,B 0,C 180,E1 19580.765,E2 19580.765} C_VEL
LIN {X 0,Y 401.43,Z 374.982,A -85,B 0,C 180,E1 19576.78,E2 19576.78} C_VEL
LIN {X 0,Y 401.43,Z 374.982,A -85,B 0,C 180,E1 19572.84,E2 19572.84} C_VEL
LIN {X 0,Y 401.438,Z 374.978,A -85,B 0,C 180,E1 19569.019,E2 19569.019} C_VEL
LIN {X 0,Y 401.455,Z 374.977,A -85,B 0,C 180,E1 19565.24,E2 19565.24} C_VEL
LIN {X 0,Y 401.47,Z 374.978,A -85,B 0,C 180,E1 19561.343,E2 19561.343} C_VEL
LIN {X 0,Y 401.475,Z 374.976,A -85,B 0,C 180,E1 19557.434,E2 19557.434} C_VEL
LIN {X 0,Y 401.474,Z 374.974,A -85,B 0,C 180,E1 19553.482,E2 19553.482} C_VEL
LIN {X 0,Y 401.455,Z 374.98,A -85,B 0,C 180,E1 19549.647,E2 19549.647} C_VEL
LIN {X 0,Y 401.442,Z 374.979,A -85,B 0,C 180,E1 19545.752,E2 19545.752} C_VEL
LIN {X 0,Y 401.43,Z 374.98,A -85,B 0,C 180,E1 19541.931,E2 19541.931} C_VEL
LIN {X 0,Y 401.425,Z 374.984,A -85,B 0,C 180,E1 19538.018,E2 19538.018} C_VEL
LIN {X 0,Y 401.425,Z 374.98,A -85,B 0,C 180,E1 19534.142,E2 19534.142} C_VEL
LIN {X 0,Y 401.424,Z 374.984,A -85,B 0,C 180,E1 19530.143,E2 19530.143} C_VEL
LIN {X 0,Y 401.431,Z 374.98,A -85,B 0,C 180,E1 19526.287,E2 19526.287} C_VEL
LIN {X 0,Y 401.441,Z 374.979,A -85,B 0,C 180,E1 19522.415,E2 19522.415} C_VEL
LIN {X 0,Y 401.454,Z 374.98,A -85,B 0,C 180,E1 19518.507,E2 19518.507} C_VEL
LIN {X 0,Y 401.478,Z 374.974,A -85,B 0,C 180,E1 19514.694,E2 19514.694} C_VEL
LIN {X 0,Y 401.471,Z 374.975,A -85,B 0,C 180,E1 19512.772,E2 19512.772} C_VEL
LIN {X 0,Y 400.524,Z 375.095,A -85,B 0,C 180,E1 19511.673,E2 19511.673} C_VEL
LIN {X 0,Y 395.901,Z 375.671,A -85,B 0,C 180,E1 19509.6,E2 19509.6} C_VEL
LIN {X 0,Y 393.641,Z 375.95,A -85,B 0,C 180,E1 19508.172,E2 19508.172} C_VEL
LIN {X 0,Y 393.489,Z 375.969,A -85,B 0,C 180,E1 19507.765,E2 19507.765} C_VEL
LIN {X 0,Y 393.497,Z 375.972,A -85,B 0,C 180,E1 19503.923,E2 19503.923} C_VEL
LIN {X 0,Y 393.512,Z 375.967,A -85,B 0,C 180,E1 19500.133,E2 19500.133} C_VEL
LIN {X 0,Y 393.531,Z 375.964,A -85,B 0,C 180,E1 19496.368,E2 19496.368} C_VEL
LIN {X 0,Y 393.536,Z 375.965,A -85,B 0,C 180,E1 19492.423,E2 19492.423} C_VEL
LIN {X 0,Y 393.532,Z 375.966,A -85,B 0,C 180,E1 19488.463,E2 19488.463} C_VEL
LIN {X 0,Y 393.526,Z 375.965,A -85,B 0,C 180,E1 19484.444,E2 19484.444} C_VEL
LIN {X 0,Y 393.516,Z 375.966,A -85,B 0,C 180,E1 19480.563,E2 19480.563} C_VEL
LIN {X 0,Y 393.505,Z 375.968,A -85,B 0,C 180,E1 19476.652,E2 19476.652} C_VEL
LIN {X 0,Y 393.497,Z 375.971,A -85,B 0,C 180,E1 19472.751,E2 19472.751} C_VEL
LIN {X 0,Y 393.493,Z 375.969,A -85,B 0,C 180,E1 19468.858,E2 19468.858} C_VEL
LIN {X 0,Y 393.488,Z 375.932,A -85,B 0,C 180,E1 19464.89,E2 19464.89} C_VEL
LIN {X 0,Y 393.492,Z 375.969,A -85,B 0,C 180,E1 19460.986,E2 19460.986} C_VEL
LIN {X 0,Y 393.494,Z 375.919,A -85,B 0,C 180,E1 19457.135,E2 19457.135} C_VEL
LIN {X 0,Y 393.504,Z 375.968,A -85,B 0,C 180,E1 19453.212,E2 19453.212} C_VEL
LIN {X 0,Y 393.512,Z 375.915,A -85,B 0,C 180,E1 19449.352,E2 19449.352} C_VEL
LIN {X 0,Y 393.535,Z 375.966,A -85,B 0,C 180,E1 19445.534,E2 19445.534} C_VEL
LIN {X 0,Y 393.527,Z 375.912,A -85,B 0,C 180,E1 19441.449,E2 19441.449} C_VEL
LIN {X 0,Y 393.536,Z 375.967,A -85,B 0,C 180,E1 19437.518,E2 19437.518} C_VEL
LIN {X 0,Y 393.539,Z 375.911,A -85,B 0,C 180,E1 19433.402,E2 19433.402} C_VEL
LIN {X 0,Y 393.534,Z 375.966,A -85,B 0,C 180,E1 19429.454,E2 19429.454} C_VEL
LIN {X 0,Y 393.535,Z 375.915,A -85,B 0,C 180,E1 19425.426,E2 19425.426} C_VEL
LIN {X 0,Y 393.534,Z 375.959,A -85,B 0,C 180,E1 19421.38,E2 19421.38} C_VEL
LIN {X 0,Y 393.524,Z 375.931,A -85,B 0,C 180,E1 19417.434,E2 19417.434} C_VEL
LIN {X 0,Y 393.508,Z 375.941,A -85,B 0,C 180,E1 19413.594,E2 19413.594} C_VEL
LIN {X 0,Y 393.501,Z 375.966,A -85,B 0,C 180,E1 19409.756,E2 19409.756} C_VEL
LIN {X 0,Y 393.494,Z 375.948,A -85,B 0,C 180,E1 19405.832,E2 19405.832} C_VEL
LIN {X 0,Y 393.493,Z 375.947,A -85,B 0,C 180,E1 19401.864,E2 19401.864} C_VEL
LIN {X 0,Y 393.552,Z 376.184,A -85,B 0,C 180,E1 19398.513,E2 19398.513} C_VEL
LIN {X 0,Y 397.734,Z 388.61,A -85,B 0,C 180,E1 19395.205,E2 19395.205} C_VEL
LIN {X 0,Y 408.975,Z 407.397,A -85,B 0,C 180,E1 19393.18,E2 19393.18} C_VEL
LIN {X 0,Y 419.541,Z 426.565,A -85,B 0,C 180,E1 19391.421,E2 19391.421} C_VEL
LIN {X 0,Y 425.306,Z 438.463,A -85,B 0,C 180,E1 19390.486,E2 19390.486} C_VEL
LIN {X 0,Y 426.239,Z 443.292,A -85,B 0,C 180,E1 19390.275,E2 19390.275} C_VEL
LIN {X 0,Y 420.044,Z 647.777,A -85,B 0,C 180,E1 19386.563,E2 19386.563} C_VEL
LIN {X 0,Y 418.638,Z 668.766,A -85,B 0,C 180,E1 19385.992,E2 19385.992} C_VEL
LIN {X 0,Y 416.798,Z 687.757,A -85,B 0,C 180,E1 19385.234,E2 19385.234} C_VEL
LIN {X 0,Y 414.935,Z 704,A -85,B 0,C 180,E1 19384.406,E2 19384.406} C_VEL
LIN {X 0,Y 412.462,Z 722.838,A -85,B 0,C 180,E1 19383.219,E2 19383.219} C_VEL
LIN {X 0,Y 409.727,Z 740.599,A -85,B 0,C 180,E1 19381.809,E2 19381.809} C_VEL
LIN {X 0,Y 407.359,Z 755.038,A -85,B 0,C 180,E1 19380.453,E2 19380.453} C_VEL
LIN {X 0,Y 404.57,Z 771.434,A -85,B 0,C 180,E1 19378.649,E2 19378.649} C_VEL
LIN {X 0,Y 401.813,Z 786.758,A -85,B 0,C 180,E1 19376.609,E2 19376.609} C_VEL
LIN {X 0,Y 399.615,Z 799.086,A -85,B 0,C 180,E1 19374.698,E2 19374.698} C_VEL
LIN {X 0,Y 397.389,Z 812.24,A -85,B 0,C 180,E1 19372.328,E2 19372.328} C_VEL
LIN {X 0,Y 395.506,Z 823.832,A -85,B 0,C 180,E1 19369.801,E2 19369.801} C_VEL
LIN {X 0,Y 394.227,Z 832.788,A -85,B 0,C 180,E1 19367.509,E2 19367.509} C_VEL
LIN {X 0,Y 393.142,Z 841.925,A -85,B 0,C 180,E1 19364.733,E2 19364.733} C_VEL
LIN {X 0,Y 392.444,Z 849.207,A -85,B 0,C 180,E1 19361.909,E2 19361.909} C_VEL
LIN {X 0,Y 392.122,Z 854.368,A -85,B 0,C 180,E1 19359.392,E2 19359.392} C_VEL
LIN {X 0,Y 391.961,Z 858.701,A -85,B 0,C 180,E1 19356.591,E2 19356.591} C_VEL
LIN {X 0,Y 391.934,Z 861.485,A -85,B 0,C 180,E1 19353.657,E2 19353.657} C_VEL
LIN {X 0,Y 391.939,Z 862.599,A -85,B 0,C 180,E1 19351.169,E2 19351.169} C_VEL
LIN {X 0,Y 391.939,Z 862.599,A -85,B 0,C 180,E1 19348.831,E2 19348.831} C_VEL
LIN {X 0,Y 391.934,Z 861.485,A -85,B 0,C 180,E1 19346.343,E2 19346.343} C_VEL
LIN {X 0,Y 391.968,Z 858.492,A -85,B 0,C 180,E1 19343.262,E2 19343.262} C_VEL
LIN {X 0,Y 392.122,Z 854.368,A -85,B 0,C 180,E1 19340.608,E2 19340.608} C_VEL
LIN {X 0,Y 392.444,Z 849.207,A -85,B 0,C 180,E1 19338.091,E2 19338.091} C_VEL
LIN {X 0,Y 393.142,Z 841.925,A -85,B 0,C 180,E1 19335.267,E2 19335.267} C_VEL
LIN {X 0,Y 394.227,Z 832.788,A -85,B 0,C 180,E1 19332.491,E2 19332.491} C_VEL
LIN {X 0,Y 395.506,Z 823.832,A -85,B 0,C 180,E1 19330.199,E2 19330.199} C_VEL
LIN {X 0,Y 397.389,Z 812.24,A -85,B 0,C 180,E1 19327.672,E2 19327.672} C_VEL
LIN {X 0,Y 399.615,Z 799.086,A -85,B 0,C 180,E1 19325.302,E2 19325.302} C_VEL
LIN {X 0,Y 401.813,Z 786.759,A -85,B 0,C 180,E1 19323.391,E2 19323.391} C_VEL
LIN {X 0,Y 404.62,Z 771.133,A -85,B 0,C 180,E1 19321.317,E2 19321.317} C_VEL
LIN {X 0,Y 407.359,Z 755.038,A -85,B 0,C 180,E1 19319.547,E2 19319.547} C_VEL
LIN {X 0,Y 409.728,Z 740.599,A -85,B 0,C 180,E1 19318.191,E2 19318.191} C_VEL
LIN {X 0,Y 412.548,Z 722.245,A -85,B 0,C 180,E1 19316.74,E2 19316.74} C_VEL
LIN {X 0,Y 414.935,Z 704,A -85,B 0,C 180,E1 19315.594,E2 19315.594} C_VEL
LIN {X 0,Y 416.798,Z 687.757,A -85,B 0,C 180,E1 19314.766,E2 19314.766} C_VEL
LIN {X 0,Y 418.732,Z 667.82,A -85,B 0,C 180,E1 19313.974,E2 19313.974} C_VEL
LIN {X 0,Y 420.071,Z 647.16,A -85,B 0,C 180,E1 19313.424,E2 19313.424} C_VEL
LIN {X 0,Y 426.244,Z 442.383,A -85,B 0,C 180,E1 19309.706,E2 19309.706} C_VEL
LIN {X 0,Y 424.678,Z 436.776,A -85,B 0,C 180,E1 19309.406,E2 19309.406} C_VEL
LIN {X 0,Y 413.873,Z 416,A -85,B 0,C 180,E1 19307.647,E2 19307.647} C_VEL
LIN {X 0,Y 403.729,Z 398.605,A -85,B 0,C 180,E1 19305.911,E2 19305.911} C_VEL
LIN {X 0,Y 397.659,Z 388.395,A -85,B 0,C 180,E1 19304.755,E2 19304.755} C_VEL
LIN {X 0,Y 394.005,Z 377.928,A -85,B 0,C 180,E1 19301.968,E2 19301.968} C_VEL
LIN {X 0,Y 393.536,Z 375.991,A -85,B 0,C 180,E1 19301.349,E2 19301.349} C_VEL
LIN {X 0,Y 393.508,Z 375.945,A -85,B 0,C 180,E1 19297.559,E2 19297.559} C_VEL
LIN {X 0,Y 393.496,Z 375.944,A -85,B 0,C 180,E1 19293.812,E2 19293.812} C_VEL
LIN {X 0,Y 393.494,Z 375.956,A -85,B 0,C 180,E1 19289.875,E2 19289.875} C_VEL
LIN {X 0,Y 393.495,Z 375.955,A -85,B 0,C 180,E1 19285.911,E2 19285.911} C_VEL
LIN {X 0,Y 393.489,Z 375.927,A -85,B 0,C 180,E1 19281.938,E2 19281.938} C_VEL
LIN {X 0,Y 393.498,Z 375.969,A -85,B 0,C 180,E1 19278.064,E2 19278.064} C_VEL
LIN {X 0,Y 393.509,Z 375.917,A -85,B 0,C 180,E1 19274.274,E2 19274.274} C_VEL
LIN {X 0,Y 393.527,Z 375.967,A -85,B 0,C 180,E1 19270.398,E2 19270.398} C_VEL
LIN {X 0,Y 393.531,Z 375.912,A -85,B 0,C 180,E1 19266.425,E2 19266.425} C_VEL
LIN {X 0,Y 393.536,Z 375.967,A -85,B 0,C 180,E1 19262.482,E2 19262.482} C_VEL
LIN {X 0,Y 393.527,Z 375.912,A -85,B 0,C 180,E1 19258.551,E2 19258.551} C_VEL
LIN {X 0,Y 393.536,Z 375.965,A -85,B 0,C 180,E1 19254.466,E2 19254.466} C_VEL
LIN {X 0,Y 393.523,Z 375.914,A -85,B 0,C 180,E1 19250.501,E2 19250.501} C_VEL
LIN {X 0,Y 393.526,Z 375.968,A -85,B 0,C 180,E1 19246.49,E2 19246.49} C_VEL
LIN {X 0,Y 393.51,Z 375.918,A -85,B 0,C 180,E1 19242.561,E2 19242.561} C_VEL
LIN {X 0,Y 393.503,Z 375.966,A -85,B 0,C 180,E1 19238.702,E2 19238.702} C_VEL
LIN {X 0,Y 393.493,Z 375.937,A -85,B 0,C 180,E1 19234.764,E2 19234.764} C_VEL
LIN {X 0,Y 393.492,Z 375.969,A -85,B 0,C 180,E1 19230.935,E2 19230.935} C_VEL
LIN {X 0,Y 393.491,Z 375.971,A -85,B 0,C 180,E1 19226.896,E2 19226.896} C_VEL
LIN {X 0,Y 393.492,Z 375.967,A -85,B 0,C 180,E1 19222.925,E2 19222.925} C_VEL
LIN {X 0,Y 393.493,Z 375.968,A -85,B 0,C 180,E1 19218.995,E2 19218.995} C_VEL
LIN {X 0,Y 393.497,Z 375.971,A -85,B 0,C 180,E1 19215.072,E2 19215.072} C_VEL
LIN {X 0,Y 393.505,Z 375.969,A -85,B 0,C 180,E1 19211.153,E2 19211.153} C_VEL
LIN {X 0,Y 393.52,Z 375.965,A -85,B 0,C 180,E1 19207.335,E2 19207.335} C_VEL
LIN {X 0,Y 393.524,Z 375.965,A -85,B 0,C 180,E1 19203.306,E2 19203.306} C_VEL
LIN {X 0,Y 393.537,Z 375.966,A -85,B 0,C 180,E1 19199.363,E2 19199.363} C_VEL
LIN {X 0,Y 393.532,Z 375.963,A -85,B 0,C 180,E1 19195.428,E2 19195.428} C_VEL
LIN {X 0,Y 393.535,Z 375.965,A -85,B 0,C 180,E1 19191.46,E2 19191.46} C_VEL
LIN {X 0,Y 393.527,Z 375.965,A -85,B 0,C 180,E1 19187.446,E2 19187.446} C_VEL
LIN {X 0,Y 393.534,Z 376.237,A -85,B 0,C 180,E1 19183.817,E2 19183.817} C_VEL
LIN {X 0,Y 394.17,Z 378.296,A -85,B 0,C 180,E1 19180.819,E2 19180.819} C_VEL
LIN {X 0,Y 395.158,Z 379.959,A -85,B 0,C 180,E1 19178.146,E2 19178.146} C_VEL
LIN {X 0,Y 396.04,Z 380.871,A -85,B 0,C 180,E1 19174.779,E2 19174.779} C_VEL
LIN {X 0,Y 396.458,Z 381.237,A -85,B 0,C 180,E1 19171.445,E2 19171.445} C_VEL
LIN {X 0,Y 396.419,Z 381.223,A -85,B 0,C 180,E1 19168.121,E2 19168.121} C_VEL
LIN {X 0,Y 395.968,Z 380.785,A -85,B 0,C 180,E1 19164.93,E2 19164.93} C_VEL
LIN {X 0,Y 395.097,Z 379.877,A -85,B 0,C 180,E1 19161.707,E2 19161.707} C_VEL
LIN {X 0,Y 394.17,Z 378.297,A -85,B 0,C 180,E1 19159.181,E2 19159.181} C_VEL
LIN {X 0,Y 393.551,Z 376.286,A -85,B 0,C 180,E1 19156.334,E2 19156.334} C_VEL
LIN {X 0,Y 393.532,Z 375.964,A -85,B 0,C 180,E1 19152.707,E2 19152.707} C_VEL
LIN {X 0,Y 393.538,Z 375.966,A -85,B 0,C 180,E1 19148.697,E2 19148.697} C_VEL
LIN {X 0,Y 393.489,Z 375.969,A -85,B 0,C 180,E1 19147.765,E2 19147.765} C_VEL
LIN {X 0,Y 392.487,Z 376.097,A -85,B 0,C 180,E1 19146.643,E2 19146.643} C_VEL
LIN {X 0,Y 386.006,Z 376.902,A -85,B 0,C 180,E1 19143.396,E2 19143.396} C_VEL
LIN {X 0,Y 385.593,Z 376.953,A -85,B 0,C 180,E1 19142.651,E2 19142.651} C_VEL
LIN {X 0,Y 385.581,Z 376.957,A -85,B 0,C 180,E1 19138.761,E2 19138.761} C_VEL
LIN {X 0,Y 385.577,Z 376.954,A -85,B 0,C 180,E1 19134.753,E2 19134.753} C_VEL
LIN {X 0,Y 385.568,Z 376.956,A -85,B 0,C 180,E1 19130.823,E2 19130.823} C_VEL
LIN {X 0,Y 385.557,Z 376.96,A -85,B 0,C 180,E1 19126.982,E2 19126.982} C_VEL
LIN {X 0,Y 385.555,Z 376.958,A -85,B 0,C 180,E1 19122.99,E2 19122.99} C_VEL
LIN {X 0,Y 385.551,Z 376.957,A -85,B 0,C 180,E1 19119.051,E2 19119.051} C_VEL
LIN {X 0,Y 385.552,Z 376.96,A -85,B 0,C 180,E1 19115.139,E2 19115.139} C_VEL
LIN {X 0,Y 385.553,Z 376.959,A -85,B 0,C 180,E1 19111.059,E2 19111.059} C_VEL
LIN {X 0,Y 385.554,Z 376.959,A -85,B 0,C 180,E1 19106.98,E2 19106.98} C_VEL
LIN {X 0,Y 385.548,Z 376.924,A -85,B 0,C 180,E1 19102.884,E2 19102.884} C_VEL
LIN {X 0,Y 385.55,Z 376.932,A -85,B 0,C 180,E1 19098.907,E2 19098.907} C_VEL
LIN {X 0,Y 385.549,Z 376.94,A -85,B 0,C 180,E1 19094.869,E2 19094.869} C_VEL
LIN {X 0,Y 385.551,Z 376.92,A -85,B 0,C 180,E1 19090.905,E2 19090.905} C_VEL
LIN {X 0,Y 385.557,Z 376.941,A -85,B 0,C 180,E1 19086.994,E2 19086.994} C_VEL
LIN {X 0,Y 385.565,Z 376.919,A -85,B 0,C 180,E1 19083.115,E2 19083.115} C_VEL
LIN {X 0,Y 385.583,Z 376.933,A -85,B 0,C 180,E1 19079.251,E2 19079.251} C_VEL
LIN {X 0,Y 385.583,Z 376.92,A -85,B 0,C 180,E1 19075.234,E2 19075.234} C_VEL
LIN {X 0,Y 385.599,Z 376.932,A -85,B 0,C 180,E1 19071.344,E2 19071.344} C_VEL
LIN {X 0,Y 385.594,Z 376.915,A -85,B 0,C 180,E1 19067.261,E2 19067.261} C_VEL
LIN {X 0,Y 385.598,Z 376.942,A -85,B 0,C 180,E1 19063.267,E2 19063.267} C_VEL
LIN {X 0,Y 385.6,Z 376.907,A -85,B 0,C 180,E1 19059.186,E2 19059.186} C_VEL
LIN {X 0,Y 385.6,Z 376.955,A -85,B 0,C 180,E1 19055.156,E2 19055.156} C_VEL
LIN {X 0,Y 385.6,Z 376.915,A -85,B 0,C 180,E1 19051.159,E2 19051.159} C_VEL
LIN {X 0,Y 385.593,Z 376.928,A -85,B 0,C 180,E1 19047.153,E2 19047.153} C_VEL
LIN {X 0,Y 385.586,Z 376.937,A -85,B 0,C 180,E1 19043.196,E2 19043.196} C_VEL
LIN {X 0,Y 385.593,Z 377.17,A -85,B 0,C 180,E1 19039.543,E2 19039.543} C_VEL
LIN {X 0,Y 389.367,Z 388.238,A -85,B 0,C 180,E1 19036.457,E2 19036.457} C_VEL
LIN {X 0,Y 400.543,Z 406.419,A -85,B 0,C 180,E1 19034.338,E2 19034.338} C_VEL
LIN {X 0,Y 411.883,Z 426.618,A -85,B 0,C 180,E1 19032.359,E2 19032.359} C_VEL
LIN {X 0,Y 419.601,Z 442.125,A -85,B 0,C 180,E1 19031.068,E2 19031.068} C_VEL
LIN {X 0,Y 420.07,Z 445.383,A -85,B 0,C 180,E1 19030.94,E2 19030.94} C_VEL
LIN {X 0,Y 413.625,Z 647.539,A -85,B 0,C 180,E1 19027.225,E2 19027.225} C_VEL
LIN {X 0,Y 412.158,Z 668.577,A -85,B 0,C 180,E1 19026.647,E2 19026.647} C_VEL
LIN {X 0,Y 410.239,Z 687.519,A -85,B 0,C 180,E1 19025.884,E2 19025.884} C_VEL
LIN {X 0,Y 408.289,Z 703.761,A -85,B 0,C 180,E1 19025.047,E2 19025.047} C_VEL
LIN {X 0,Y 405.69,Z 722.701,A -85,B 0,C 180,E1 19023.838,E2 19023.838} C_VEL
LIN {X 0,Y 402.834,Z 740.359,A -85,B 0,C 180,E1 19022.419,E2 19022.419} C_VEL
LIN {X 0,Y 400.36,Z 754.684,A -85,B 0,C 180,E1 19021.057,E2 19021.057} C_VEL
LIN {X 0,Y 397.519,Z 770.561,A -85,B 0,C 180,E1 19019.288,E2 19019.288} C_VEL
LIN {X 0,Y 394.491,Z 786.516,A -85,B 0,C 180,E1 19017.143,E2 19017.143} C_VEL
LIN {X 0,Y 392.168,Z 798.843,A -85,B 0,C 180,E1 19015.199,E2 19015.199} C_VEL
LIN {X 0,Y 389.797,Z 811.997,A -85,B 0,C 180,E1 19012.787,E2 19012.787} C_VEL
LIN {X 0,Y 387.763,Z 823.731,A -85,B 0,C 180,E1 19010.177,E2 19010.177} C_VEL
LIN {X 0,Y 386.443,Z 832.341,A -85,B 0,C 180,E1 19007.932,E2 19007.932} C_VEL
LIN {X 0,Y 385.264,Z 841.518,A -85,B 0,C 180,E1 19005.099,E2 19005.099} C_VEL
LIN {X 0,Y 384.492,Z 848.967,A -85,B 0,C 180,E1 19002.159,E2 19002.159} C_VEL
LIN {X 0,Y 384.141,Z 854.129,A -85,B 0,C 180,E1 18999.589,E2 18999.589} C_VEL
LIN {X 0,Y 383.968,Z 858.463,A -85,B 0,C 180,E1 18996.729,E2 18996.729} C_VEL
LIN {X 0,Y 383.936,Z 861.248,A -85,B 0,C 180,E1 18993.733,E2 18993.733} C_VEL
